(*Gestion des consigne de pompage procédé*)
IF RQ_MARCHE_POMPAGE_PROC OR RQ_MARCHE_REGUL_GAZ[1] OR RQ_MARCHE_REGUL_GAZ[2] THEN
	CONS_MODE := PRM_MODE_PUMPING;
	CONS_PRESSURE := PRM_PR_PUMPING;
	CONS_POSITION := PRM_POS_PUMPING;
	CONS_HI_PRESSURE := PRM_PR_HI_PUMPING;
	CONS_LOW_PRESSURE := PRM_PR_LO_PUMPING;
	CONS_TIM_PRESSURE :=  REAL_TO_TIME ( PRM_TIM_PR_PUMPING * 1000);
END_IF

(*Gestion de la consigne pour la ligne de gaz n°1*)
IF RQ_MARCHE_GAZ[1] THEN
	CONS_FLOW_GAZ_1 := PRM_FLOW_GAZ1;
END_IF

(*Gestion de la consigne pour la ligne de gaz n°2*)
IF RQ_MARCHE_GAZ[2] THEN
	CONS_FLOW_GAZ_2 := PRM_FLOW_GAZ2;
END_IF

(*Demande d'arrêt des sources, que si source pas démarrée pour anticipation*)
RQ_STOP_EVAP_S1 := (FM_ETAPE14.Q AND NOT PRM_UTIL_SOURCE1_ANT) OR (FM_ETAPE10.Q AND NOT PRM_UTIL_SOURCE1);
RQ_STOP_EVAP_S2 := (FM_ETAPE14.Q AND NOT PRM_UTIL_SOURCE2_ANT) OR (FM_ETAPE10.Q AND NOT PRM_UTIL_SOURCE2);
RQ_STOP_EVAP_S3 := (FM_ETAPE14.Q AND NOT PRM_UTIL_SOURCE3_ANT) OR (FM_ETAPE10.Q AND NOT PRM_UTIL_SOURCE3);
RQ_STOP_EVAP_S4 := (FM_ETAPE14.Q AND NOT PRM_UTIL_SOURCE4_ANT) OR (FM_ETAPE10.Q AND NOT PRM_UTIL_SOURCE4);


(*Mise à jour du temps de préparation pour les couches anticipées :
remarque dans le cas de plusieurs sources, elles doivent toutes avoir le même temps de prépa (cf. editeur), mais on prend le max pour sécu*)
IF PRM_UTIL_SOURCE1_ANT THEN
	VAR_TPS_PREPA_ANT1 := PRM_TPS_PREPA_SOURCE1;
	VAR_TPS_PREPA_ANT1_2s := VAR_TPS_PREPA_ANT1 + 5;
ELSE
	VAR_TPS_PREPA_ANT1 := 0;
	VAR_TPS_PREPA_ANT1_2s := 0;
END_IF
IF PRM_UTIL_SOURCE2_ANT THEN
	VAR_TPS_PREPA_ANT2 := PRM_TPS_PREPA_SOURCE2;
	VAR_TPS_PREPA_ANT2_2s := VAR_TPS_PREPA_ANT2 + 5;
ELSE
	VAR_TPS_PREPA_ANT2 := 0;
	VAR_TPS_PREPA_ANT2_2s := 0;
END_IF
IF PRM_UTIL_SOURCE3_ANT THEN
	VAR_TPS_PREPA_ANT3 := PRM_TPS_PREPA_SOURCE3;
	VAR_TPS_PREPA_ANT3_2s := VAR_TPS_PREPA_ANT3 + 5;
ELSE
	VAR_TPS_PREPA_ANT3 := 0;
	VAR_TPS_PREPA_ANT3_2s := 0;
END_IF
IF PRM_UTIL_SOURCE4_ANT THEN
	VAR_TPS_PREPA_ANT4 := PRM_TPS_PREPA_SOURCE4;
	VAR_TPS_PREPA_ANT4_2s := VAR_TPS_PREPA_ANT4 + 5;
ELSE
	VAR_TPS_PREPA_ANT4 := 0;
	VAR_TPS_PREPA_ANT4_2s := 0;
END_IF

(*
(*Les nouvelles épaisseurs se trouvent dans le tableau*)
PRM_EPAISSEUR:= PRM_NEW_EPAISSEUR[STATE_LAYER];
*)

(*calcul du temps restant : version avec vitesse aggrégée théorique (somme des vitesses ds sources utilisées dans l'étape en cours)*)
(*calcul vitesse théorique*)
IF FM_ETAPE12.Q THEN
	VAR_CALCUL_VITESSE_THEORIQUE := PRM_SOURCE1_RATE * BOOL_TO_INT(PRM_UTIL_SOURCE1) +
										PRM_SOURCE2_RATE * BOOL_TO_INT(PRM_UTIL_SOURCE2) +
										PRM_SOURCE3_RATE * BOOL_TO_INT(PRM_UTIL_SOURCE3) +
										PRM_SOURCE4_RATE * BOOL_TO_INT(PRM_UTIL_SOURCE4);
ELSIF OP_RUN.Etape.4 THEN
	VAR_CALCUL_VITESSE_THEORIQUE := 0;
END_IF
IF VAR_CALCUL_VITESSE_THEORIQUE <> 0 THEN
	VAR_TPS_RESTANT_DEPOT := REAL_TO_INT((PRM_EPAISSEUR - I_Global_Thick) / VAR_CALCUL_VITESSE_THEORIQUE);
END_IF


(*temporisation de lissage du bagotage de la vitesse aggrégée si PID pas top, on doit rester inférieur plus de 2s pour lancer la prépa anticipée*)
TIMER_Lancement_Ant_S1.PT := T#1s;
TIMER_Lancement_Ant_S1.IN := (VAR_TPS_RESTANT_DEPOT <= VAR_TPS_PREPA_ANT1_2s) AND TIMER_RAZ_THICKNESS.Q;
TIMER_Lancement_Ant_S1();

TIMER_Lancement_Ant_S2.PT := T#1s;
TIMER_Lancement_Ant_S2.IN := (VAR_TPS_RESTANT_DEPOT <= VAR_TPS_PREPA_ANT2_2s) AND TIMER_RAZ_THICKNESS.Q;
TIMER_Lancement_Ant_S2();

TIMER_Lancement_Ant_S3.PT := T#1s;
TIMER_Lancement_Ant_S3.IN := (VAR_TPS_RESTANT_DEPOT <= VAR_TPS_PREPA_ANT3_2s) AND TIMER_RAZ_THICKNESS.Q;
TIMER_Lancement_Ant_S3();

TIMER_Lancement_Ant_S4.PT := T#1s;
TIMER_Lancement_Ant_S4.IN := (VAR_TPS_RESTANT_DEPOT <= VAR_TPS_PREPA_ANT4_2s) AND TIMER_RAZ_THICKNESS.Q;
TIMER_Lancement_Ant_S4();

(*Lancement de la prépa anticipée seulement si pas de Quartz sous le cache source*)
FM_Prepa_Ant_S1.CLK := 	OP_RUN.Etape.12 AND TIMER_RAZ_THICKNESS.Q AND
						PRM_UTIL_SOURCE1_ANT AND NOT PRM_CTRL_DELAY_SOURCE1 AND
						TIMER_Lancement_Ant_S1.Q;
						(*VAR_TPS_RESTANT_DEPOT <= VAR_TPS_PREPA_ANT1_2s;*)

FM_Prepa_Ant_S2.CLK := 	OP_RUN.Etape.12 AND TIMER_RAZ_THICKNESS.Q AND
						PRM_UTIL_SOURCE2_ANT  AND NOT PRM_CTRL_DELAY_SOURCE2 AND
						TIMER_Lancement_Ant_S2.Q;
						(*VAR_TPS_RESTANT_DEPOT <= VAR_TPS_PREPA_ANT2_2s;*)

FM_Prepa_Ant_S3.CLK := 	OP_RUN.Etape.12 AND TIMER_RAZ_THICKNESS.Q AND
						PRM_UTIL_SOURCE3_ANT AND NOT PRM_CTRL_DELAY_SOURCE3 AND
						TIMER_Lancement_Ant_S3.Q;
						(*VAR_TPS_RESTANT_DEPOT <= VAR_TPS_PREPA_ANT3_2s;*)

FM_Prepa_Ant_S4.CLK := 	OP_RUN.Etape.12 AND TIMER_RAZ_THICKNESS.Q AND
						PRM_UTIL_SOURCE4_ANT AND NOT PRM_CTRL_DELAY_SOURCE4 AND
						TIMER_Lancement_Ant_S4.Q;
						(*VAR_TPS_RESTANT_DEPOT <= VAR_TPS_PREPA_ANT4_2s;*)

FM_Prepa_Ant_S1();
FM_Prepa_Ant_S2();
FM_Prepa_Ant_S3();
FM_Prepa_Ant_S4();


(*Demande de préparation : soit étape 8 sur couche classique (mais pas dans le cas ou elle a été anticipée), soit FM de go anticipation
	(mais que si la source est en étape 0 ou en étape 16, cad arrétée ou cloture finie (sinon le RQ_Evap tombe à l'eau) 
remarque : dans ce cas le var_prepa_lancée est peut etre redondant 

Pas de demande d'anticipation s'il y a un Quartz d'étalonnage de la vitesse de dépôt sous le cache source*)
RQ_PREP_S1 := (FM_ETAPE10.Q AND PRM_UTIL_SOURCE1 AND NOT PRM_ANTICIPATION_COUCHE)
					OR (FM_Prepa_Ant_S1.Q AND NOT  VAR_Prepa_S1_Lancee AND NOT PRM_CTRL_DELAY_SOURCE1
						AND I_SOURCE1_ARRET );

RQ_PREP_S2 := (FM_ETAPE10.Q AND PRM_UTIL_SOURCE2 AND NOT PRM_ANTICIPATION_COUCHE)
					OR (FM_Prepa_Ant_S2.Q AND NOT VAR_Prepa_S2_Lancee AND NOT PRM_CTRL_DELAY_SOURCE2
						AND I_SOURCE2_ARRET);

RQ_PREP_S3 := (FM_ETAPE10.Q AND PRM_UTIL_SOURCE3 AND NOT PRM_ANTICIPATION_COUCHE)
					OR (FM_Prepa_Ant_S3.Q AND NOT VAR_Prepa_S3_Lancee AND NOT PRM_CTRL_DELAY_SOURCE3
						AND I_SOURCE3_ARRET);

RQ_PREP_S4 := (FM_ETAPE10.Q AND PRM_UTIL_SOURCE4 AND NOT PRM_ANTICIPATION_COUCHE)
					OR (FM_Prepa_Ant_S4.Q AND NOT VAR_Prepa_S4_Lancee AND NOT PRM_CTRL_DELAY_SOURCE4
						AND I_SOURCE4_ARRET);



(*variable mise à 1 au premier front montant pour éviter de relancer la prépa si bagotage du temps restant de dépot, remis à 0 en 6 cad apres lecture couche suivante*)
IF FM_Prepa_Ant_S1.Q THEN
	VAR_Prepa_S1_Lancee := TRUE;
ELSIF OP_RUN.Etape.6 OR OP_RUN.Etape.0 THEN
	VAR_Prepa_S1_Lancee := FALSE;
END_IF

IF FM_Prepa_Ant_S2.Q THEN
	VAR_Prepa_S2_Lancee := TRUE;
ELSIF OP_RUN.Etape.6 OR OP_RUN.Etape.0 THEN
	VAR_Prepa_S2_Lancee := FALSE;
END_IF

IF FM_Prepa_Ant_S3.Q THEN
	VAR_Prepa_S3_Lancee := TRUE;
ELSIF OP_RUN.Etape.6 OR OP_RUN.Etape.0 THEN
	VAR_Prepa_S3_Lancee := FALSE;
END_IF

IF FM_Prepa_Ant_S4.Q THEN
	VAR_Prepa_S4_Lancee := TRUE;
ELSIF OP_RUN.Etape.6 OR OP_RUN.Etape.0 THEN
	VAR_Prepa_S4_Lancee := FALSE;
END_IF


(*Lancement évaporation*)
RQ_EVAP_S1 := OP_RUN.Etape.12 AND PRM_UTIL_SOURCE1;
RQ_EVAP_S2 := OP_RUN.Etape.12 AND PRM_UTIL_SOURCE2;
RQ_EVAP_S3 := OP_RUN.Etape.12 AND PRM_UTIL_SOURCE3;
RQ_EVAP_S4 := OP_RUN.Etape.12 AND PRM_UTIL_SOURCE4;

(*Défaut de lecture d'une étape*)
DEF_READ_LAYER.VAL1 := UINT_TO_STRING(STATE_LAYER);
DEF_READ_LAYER.CONDITION := OP_RUN.Etape.20;
DEF_READ_LAYER();

(*Défaut de lecture d'une étape anticipée*)
DEF_READ_LAYER_ANT.VAL1 := UINT_TO_STRING(STATE_LAYER + 1);
DEF_READ_LAYER_ANT.CONDITION := OP_RUN.Etape.21;
DEF_READ_LAYER_ANT();

(*Défaut time out programmation XTC*)
DEF_PROG_QZ.CONDITION := OP_RUN.Etape.9;
DEF_PROG_QZ.DELAY := T#45s;
DEF_PROG_QZ();

(*Défaut time out raz epaisseur controleur XTC*)
DEF_RAZ_QZ.CONDITION := OP_RUN.Etape.11;
DEF_RAZ_QZ.DELAY := T#20s;
DEF_RAZ_QZ();

(*Défaut de passage en STOP du contrôleur de dépôt pendant l'évaporation*)
DEF_CONTROLLER_STOPPED.CONDITION := OP_RUN.Etape.12 AND I_CONTROLEUR_PHASE = 'Deposit' AND  I_Controleur_Stopped;
DEF_CONTROLLER_STOPPED.DELAY:= T#20s;
DEF_CONTROLLER_STOPPED();

(*
(*Défaut de panne quartz générale*)
DEF_QF.CONDITION := I_PC_QUARTZ.STATE_Qz_general_failure AND NOT OP_RUN.Etape.0;
DEF_QF.VAL1 := USINT_TO_STRING(I_PC_QUARTZ.STATE_QF_code);
DEF_QF;
*)

(*reset des ordres*)
IF RCP_NEXT_LAYER AND M_NEXT_LAYER THEN
	M_NEXT_LAYER:=FALSE;
END_IF;


STATE_RATE_AGREGATE := I_Global_Rate;			(*vitesse globale renvoyé par le contrôleur*)
STATE_THICKNESS_AGREGATE  := I_Global_Thick;	(*epaisseur globale renvoyé par le contrôleur*)

STATE_END_OF_LAYER := OP_RUN.Etape.13;
STATE_EVAP := OP_RUN.Etape.12;

IF OP_RUN.Etape.17 THEN
	VAR_Loop_In_Process:= TRUE;
ELSIF OP_RUN.Etape.4 THEN
	VAR_Loop_In_Process:= FALSE;
END_IF

(*Sorties contrôleur*)
OUT_RAZ_THICK_CONTROLEUR:= OP_RUN.Etape.11 AND (NOT I_MODE_REPRISE OR NOT VAR_MEM_LAYER_INTERRUPTED) AND NOT VAR_MEM_COUCHE_TERMINEE;
OUT_RESET_CONTROLEUR:= OP_RUN.Etape.3;
OUT_STOP_CONTROLEUR:= OP_RUN.Etape.2 OR OP_RUN.Etape.13;


IF  OP_RUN.Etape.10 AND (NOT I_MODE_REPRISE OR NOT VAR_MEM_LAYER_INTERRUPTED) THEN
	VAR_MEM_RAZ_THICKNESS := FALSE;
END_IF;
TIMER_RAZ_THICKNESS.PT := T#3s;
TIMER_RAZ_THICKNESS.IN := VAR_MEM_RAZ_THICKNESS;
TIMER_RAZ_THICKNESS();

ACTION RUN_PROCESS:
(*GRAFCET EXECUTION PROCEDE*)
(* initialisation du grafcet*)

OP_RUN(
	N_STEP_OP_OK:=15,
	N_STEP_OP_NOK:= 0);

(* initialisation du grafcet*)
IF 		OP_RUN.Etape = 0 THEN
				OP_RUN.Etape.0 := TRUE;
(*repositionnement sur étape 0*)
ELSIF  NOT I_ON THEN
				OP_Run.Etape:= 0;			(*RAZ grafcet*)
				OP_Run.Etape.0:=TRUE;
(*Repositionnement sur demande fin de couche*)
ELSIF (OP_RUN.Etape.6 OR OP_RUN.Etape.7 OR OP_RUN.Etape.9 OR OP_RUN.Etape.10 OR OP_RUN.Etape.11 OR OP_RUN.Etape.12) AND
		(RCP_NEXT_LAYER)  THEN
				(*si evaporation en cours sur les sources*)
				IF  (OP_RUN.Etape.10 OR OP_RUN.Etape.11 OR OP_RUN.Etape.12) THEN
					RQ_NEXT_LAYER := TRUE; 	(*demande de fin de couche au bloc de gestion des sources*)
				END_IF
				I_MODE_REPRISE := FALSE;
				VAR_MEM_COUCHE_TERMINEE := TRUE;
				(*VAR_Cpt_Boucle:=1;*)	(*RAZ du compteur de boucle*)
				OP_RUN.Etape := 0;
				OP_RUN.Etape.13 := TRUE;
(*étape 0-1 attente ordre execution de l'empilement*)
ELSIF OP_RUN.etape.0 AND I_ON THEN
				OP_RUN.Etape.1 	:=TRUE;
				OP_RUN.Etape.0 	:=FALSE;
(*étape 1-2 *)
ELSIF	OP_RUN.Etape.1 AND NOT I_MODE_REPRISE THEN
				VAR_MEM_LAYER_INTERRUPTED  := FALSE;
				VAR_MEM_COUCHE_TERMINEE := FALSE;
				VAR_MEM_PREP_OPT_TERMINEE := FALSE;
				VAR_Cpt_Boucle:= 1;
				STATE_LAYER:= 1;
				OP_RUN.Etape.2:=TRUE;
				OP_RUN.Etape.1:=FALSE;
(*étape 1-2*)
ELSIF OP_RUN.Etape.1 AND
				(NOT VAR_MEM_LAYER_INTERRUPTED AND I_MODE_REPRISE)
				THEN (*STOP et RESET si mode reprise et pas couche interrompue*)
				OP_RUN.Etape.2:= TRUE;
				OP_RUN.Etape.1:= FALSE;
(*étape 1-4 *)
ELSIF	OP_RUN.Etape.1 AND
				(VAR_MEM_LAYER_INTERRUPTED  AND I_MODE_REPRISE)
				THEN (*Pas de STOP ni de RESET si mode reprise et couche interrompue*)
				OP_RUN.Etape.4:=TRUE;
				OP_RUN.Etape.1:=FALSE;

(*etape 2-3*)
ELSIF OP_RUN.Etape.2  AND TIMER_Stop_Controller.Q(*AND I_ACTION_CONTROLEUR_OK*) THEN
				OP_RUN.Etape.3:=TRUE;
				OP_RUN.Etape.2:=FALSE;

(*etape 3-4*)
ELSIF OP_RUN.Etape.3
				AND TIMER_Reset_Controller.Q (*AND I_ACTION_CONTROLEUR_OK*) AND I_CONTROLEUR_PHASE = 'Ready' THEN		(*IC6 à l'état READY si la RAZ empilement à été effectué *)
				OP_RUN.Etape.4:=TRUE;
				OP_RUN.Etape.3	:=FALSE;

(*etape 4-20*)
ELSIF OP_RUN.Etape.4 AND
				(TIMER_TIMEOUT.Q OR I_LAYER_LOADING_NOK) THEN
				OP_RUN.Etape.20:=TRUE;
				OP_RUN.Etape.4	:=FALSE;

(*etape 4-5*)
ELSIF OP_RUN.Etape.4 AND I_LAYER_LOADING_OK THEN
				OP_RUN.Etape.5		:=TRUE;
				OP_RUN.Etape.4		:=FALSE;

(*etape 5-21*)
ELSIF OP_RUN.Etape.5 AND
				(TIMER_TIMEOUT_ANT.Q OR I_LAYER_ANT_LOADING_NOK) THEN
				OP_RUN.Etape.21 := TRUE;
				OP_RUN.Etape.5 := FALSE;

(*etape 5-6*)
ELSIF OP_RUN.Etape.5 AND (I_LAYER_ANT_LOADING_OK OR I_NO_MORE_LAYER_ANT) THEN	(*Couche anticipée chargé ou pas de couche anticipée*)
				OP_RUN.Etape.6 := TRUE;
				OP_RUN.Etape.5 := FALSE;

(*etape 6-7*)
ELSIF OP_RUN.Etape.6 AND
				((I_ROTATION_PS_OK AND NOT I_NO_ROTATION_PS) OR (I_STOP_ROT_PS_OK AND I_NO_ROTATION_PS))
				AND ((I_STOP_TILT_PS_OK AND I_MODE_TILT = 2) OR (I_MODE_TILT = 1))
				AND I_DOME_IN_POSITION
				AND (
				(I_MARCHE_CHAUFFAGE_OK AND (PRM_MODE_CHAUFFAGE = 1)
						AND (I_STAB_CHAUFFAGE_OK OR NOT PRM_WAIT_STAB_TEMP)
				 )
				OR
				(I_ARRET_CHAUFFAGE_OK AND (PRM_MODE_CHAUFFAGE = 0))
				OR (PRM_MODE_CHAUFFAGE = 2)
				)
				AND(( I_ARRET_GAZ1_OK OR VAR_Util_Gaz[1]) AND (I_ARRET_GAZ2_OK OR VAR_Util_Gaz[2]))
				THEN
				OP_RUN.Etape.7:=TRUE;
				OP_RUN.Etape.6:= FALSE;

(*etape 7-9*)
ELSIF OP_RUN.Etape.7 AND (
				(I_MARCHE_IAD_OK AND PRM_OP_UTIL_IAD) OR
				(I_ARRET_IAD_OK AND NOT PRM_OP_UTIL_IAD) OR NOT CONF_IAD
				)
				AND I_TILT_PS_OK
				AND NOT I_MODE_REPRISE
				THEN
				OP_RUN.Etape.9:=TRUE;
				OP_RUN.Etape.7:=FALSE;

(*etape 7-10 - On ne recharge pas les paramètres dans l'XTC en cas de reprise*)
ELSIF OP_RUN.Etape.7 AND (
				(I_MARCHE_IAD_OK AND PRM_OP_UTIL_IAD) OR
				(I_ARRET_IAD_OK AND NOT PRM_OP_UTIL_IAD) OR NOT CONF_IAD
				)
				AND I_TILT_PS_OK
				AND I_MODE_REPRISE
				THEN
				OP_RUN.Etape.10:=TRUE;
				OP_RUN.Etape.7:=FALSE;

(*Etape 9-10*)
ELSIF OP_RUN.Etape.9 AND I_PROG_CONTROLEUR_OK THEN		(*Programmation contrôleur ok*)
				OP_RUN.Etape.10:=TRUE;
				OP_RUN.Etape.9:=FALSE;

(*Etape 10-11*)
ELSIF OP_RUN.Etape.10
	    AND (I_PREP_SOURCE1_OK OR (NOT PRM_UTIL_SOURCE1 AND I_STOP_EVAP1_OK))
	    AND (I_PREP_SOURCE2_OK OR (NOT PRM_UTIL_SOURCE2 AND I_STOP_EVAP2_OK))
	    AND (I_PREP_SOURCE3_OK OR (NOT PRM_UTIL_SOURCE3 AND I_STOP_EVAP3_OK))
	    AND (I_PREP_SOURCE4_OK OR (NOT PRM_UTIL_SOURCE4 AND I_STOP_EVAP4_OK))
	THEN
				OP_RUN.Etape.11:=TRUE;
				OP_RUN.Etape.10:=FALSE;

(*Demande RAZ épaisseur si pas de mode reprise*)
(*Etape 11-12*)
ELSIF OP_RUN.Etape.11  AND
				(*On vérifie que l'épaisseur à bien été remis à 0*)
				((I_Global_Thick <= 0.1) OR
				(VAR_MEM_LAYER_INTERRUPTED  AND I_MODE_REPRISE) OR
				(VAR_MEM_COUCHE_TERMINEE AND I_MODE_REPRISE)
				)
				AND TIMER_RAZ_EPAISSEUR.Q
				THEN
				(*on déclenche la temporisation aprés RAZ épaisseur*)
				IF (I_Global_Thick<= 0.1) THEN
					VAR_MEM_RAZ_THICKNESS := TRUE;
				END_IF
				VAR_MEM_LAYER_INTERRUPTED := TRUE;
				OP_RUN.Etape.12:=TRUE;
				OP_RUN.Etape.11:=FALSE;

(*Etape 12-13 épaisseur atteinte et tempo de validation de remise à 0 de l'épaisseur*)
ELSIF OP_RUN.Etape.12  AND
			((I_END_DEPOT OR VAR_MEM_COUCHE_TERMINEE) AND TIMER_RAZ_THICKNESS.Q) THEN
				I_MODE_REPRISE := FALSE;
				VAR_MEM_LAYER_INTERRUPTED := FALSE;
				VAR_MEM_COUCHE_TERMINEE := TRUE;
				OP_RUN.Etape.13:=TRUE;
				OP_RUN.Etape.12:=FALSE;

(*Cloture des sources*)
(*Etape 13-16*)
ELSIF OP_RUN.Etape.13
	    AND (I_CLOT_SOURCE1_OK OR NOT PRM_UTIL_SOURCE1
				OR PRM_UTIL_SOURCE1_ANT OR PRM_UTIL_SOURCE2_ANT OR PRM_UTIL_SOURCE3_ANT OR PRM_UTIL_SOURCE4_ANT)
	    AND (I_CLOT_SOURCE2_OK OR NOT PRM_UTIL_SOURCE2
				OR PRM_UTIL_SOURCE1_ANT OR PRM_UTIL_SOURCE2_ANT OR PRM_UTIL_SOURCE3_ANT OR PRM_UTIL_SOURCE4_ANT)
	    AND (I_CLOT_SOURCE3_OK OR NOT PRM_UTIL_SOURCE3
				OR PRM_UTIL_SOURCE1_ANT OR PRM_UTIL_SOURCE2_ANT OR PRM_UTIL_SOURCE3_ANT OR PRM_UTIL_SOURCE4_ANT)
	    AND (I_CLOT_SOURCE4_OK OR NOT PRM_UTIL_SOURCE4
				OR PRM_UTIL_SOURCE1_ANT OR PRM_UTIL_SOURCE2_ANT OR PRM_UTIL_SOURCE3_ANT OR PRM_UTIL_SOURCE4_ANT)
	    AND (((I_ARRET_REGUL_GAZ_OK[1] AND I_MARCHE_POMPAGE_SEC_OK)  OR NOT (PRM_MODE_PUMPING = 2)) OR ((I_ARRET_REGUL_GAZ_OK[2] AND I_MARCHE_POMPAGE_SEC_OK)  OR NOT (PRM_MODE_PUMPING = 3)))
		THEN
				STATE_LAYER := STATE_LAYER +1;
				(*RAZ des flags*)
				VAR_MEM_LAYER_INTERRUPTED := FALSE;
				VAR_MEM_COUCHE_TERMINEE := FALSE;
				OP_RUN.Etape.16:=TRUE;
				OP_RUN.Etape.13:=FALSE;

(*Boucle à effectuer*)
(*Etape 16-17*)
ELSIF OP_RUN.Etape.16
		AND (PRM_LOOP AND ((STATE_LAYER = PRM_LOOP_LAST_LAYER +1) AND (VAR_Cpt_Boucle < PRM_NB_LOOP)))
			THEN
				STATE_LAYER := PRM_LOOP_FIRST_LAYER;
				VAR_Cpt_Boucle:= VAR_Cpt_Boucle + 1;
				OP_RUN.Etape.17:= TRUE;
				OP_RUN.Etape.16:= FALSE;

(*Pas de boucle à effectuer ou nombre de boucle OK*)
(*Etape 16-2*)
ELSIF OP_RUN.Etape.16
		AND ( NOT PRM_LOOP OR NOT (VAR_Cpt_Boucle > PRM_NB_LOOP))  THEN
				OP_RUN.Etape.2	:= TRUE;
				OP_RUN.Etape.16	:= FALSE;
(*
(*Chargement du numéro de couche de départ*)
(*Etape 17-6*)
ELSIF OP_RUN.Etape.17
		AND I_LAYER_LOADING_OK THEN
				OP_RUN.Etape.6:= TRUE;
				OP_RUN.Etape.17:= FALSE;
*)
(*
(*Etape 17-20*)
ELSIF OP_RUN.Etape.17 AND
		(TIMER_TIMEOUT.Q OR I_LAYER_LOADING_NOK) THEN
				OP_RUN.Etape.20:= TRUE;
				OP_RUN.Etape.17:= FALSE;
*)

(*Etape 17-2*)
ELSIF OP_RUN.Etape.17 THEN
				OP_RUN.Etape.2:=TRUE;
				OP_RUN.Etape.17:=FALSE;
(*Etape 4-14*)
ELSIF OP_RUN.Etape.4 AND  I_NO_MORE_LAYER THEN
				OP_RUN.Etape.14:=TRUE;
				OP_RUN.Etape.4:=FALSE;

(*Etape 14-15*)
ELSIF OP_RUN.Etape.14 AND  I_STOP_EVAP1_OK AND I_STOP_EVAP2_OK AND I_STOP_EVAP3_OK
		AND I_DOME_IN_POSITION
		AND I_STOP_ROT_PS_OK
		AND I_STOP_TILT_PS_OK
		AND I_ARRET_REGUL_GAZ_OK[1]
		AND I_ARRET_REGUL_GAZ_OK[2]
		AND I_MARCHE_POMPAGE_SEC_OK
		AND I_STOP_EVAP4_OK  AND I_ARRET_GAZ1_OK AND I_ARRET_GAZ2_OK
		AND (I_ARRET_IAD_OK OR NOT CONF_IAD) THEN
				OP_RUN.Etape.15:=TRUE;
				OP_RUN.Etape.14:=FALSE;
END_IF

OP_RUN.POST();
END_ACTION

END_FUNCTION_BLOCK

// ---- POUs/Fonction/FONCTION MODEMARCHE/BLOCK_STEP_BOUCLE.TcPOU
FUNCTION_BLOCK BLOCK_STEP_BOUCLE

VAR_INPUT
	RESET:							BOOL;
	I_ON:							BOOL;
	I_CURRENT_STEP:					UINT;
	PRM_ITER_BOUCLE:				USINT;
	PRM_ETAPE_BOUCLE:				UINT;
END_VAR

VAR_OUTPUT
	STATE_OK:						BOOL;
	AUTOR_STEP:						BOOL;
	STATE_ITER_BOUCLE:				USINT;
	O_NEXT_STEP:					UINT;
	RQ_BOUCLE:						BOOL;
	RQ_SAUT:						BOOL;
END_VAR

VAR
	MEM_BOUCLE:						BOOL;
	MEM_START_BOUCLE:				UINT;
	MEM_STOP_BOUCLE:				UINT;
	FM_ON:							R_TRIG;
END_VAR

(*Autorisation*)
AUTOR_STEP	:=	( (PRM_ITER_BOUCLE = 0) AND (PRM_ETAPE_BOUCLE > I_CURRENT_STEP) ) (*saut sur étape après*)
					OR
					( (PRM_ITER_BOUCLE > 0) AND (PRM_ETAPE_BOUCLE < I_CURRENT_STEP) ) (*boucle sur étape avant*)
					OR
					( NOT MEM_BOUCLE AND ((MEM_START_BOUCLE <> I_CURRENT_STEP) OR (MEM_STOP_BOUCLE <> PRM_ETAPE_BOUCLE)) ); (*pas 2 boucles imbriquées*)

(*Reset fonction hors procédé*)
IF RESET THEN
	MEM_BOUCLE			:=	FALSE;
	MEM_START_BOUCLE	:=	0;
	MEM_STOP_BOUCLE		:=	0;
	STATE_ITER_BOUCLE	:=	0;
	O_NEXT_STEP			:=	0;
	RQ_BOUCLE				:=	FALSE;
	RQ_SAUT				:=	FALSE;
	STATE_OK				:=	FALSE;
END_IF

IF NOT I_ON THEN
	STATE_OK				:=	FALSE;
	RQ_BOUCLE				:=	FALSE;
	RQ_SAUT				:=	FALSE;
END_IF

(*Front montant*)
FM_ON.CLK	:=	I_ON;
FM_ON();

IF FM_ON.Q THEN
	(*Gestion saut*)
	IF PRM_ITER_BOUCLE = 0 THEN
		MEM_BOUCLE			:=	FALSE;
		MEM_START_BOUCLE	:=	0;
		MEM_STOP_BOUCLE		:=	0;
		STATE_ITER_BOUCLE	:=	0;
		O_NEXT_STEP			:=	PRM_ETAPE_BOUCLE;
		RQ_SAUT				:=	TRUE;
		STATE_OK				:=	TRUE;

	(*Gestion boucle*)
	ELSE
		(*Départ boucle*)
		IF MEM_BOUCLE = 0THEN
			MEM_BOUCLE			:=	TRUE;
			MEM_START_BOUCLE	:=	I_CURRENT_STEP;
			MEM_STOP_BOUCLE		:=	PRM_ETAPE_BOUCLE;
			STATE_ITER_BOUCLE	:=	1;
			O_NEXT_STEP			:=	PRM_ETAPE_BOUCLE;
			RQ_BOUCLE				:=	TRUE;
			STATE_OK				:=	TRUE;
		ELSE
			(*Fin boucle*)
			IF MEM_BOUCLE AND (STATE_ITER_BOUCLE >= PRM_ITER_BOUCLE) THEN
				MEM_BOUCLE			:=	FALSE;
				MEM_START_BOUCLE	:=	0;
				MEM_STOP_BOUCLE		:=	0;
				STATE_ITER_BOUCLE	:=	0;
				O_NEXT_STEP			:=	I_CURRENT_STEP + 1;
				STATE_OK				:=	TRUE;
			(*Suite boucle*)
			ELSE
				MEM_BOUCLE			:=	TRUE;
				MEM_START_BOUCLE	:=	I_CURRENT_STEP;
				MEM_STOP_BOUCLE		:=	PRM_ETAPE_BOUCLE;
				STATE_ITER_BOUCLE	:=	STATE_ITER_BOUCLE + 1;
				O_NEXT_STEP			:=	MEM_STOP_BOUCLE;
				RQ_BOUCLE				:=	TRUE;
				STATE_OK				:=	TRUE;
			END_IF
		END_IF
	END_IF
END_IF

END_FUNCTION_BLOCK

// ---- POUs/Fonction/FONCTIONS PUISSANCE/BLOCK_CPT_USURE.TcPOU
FUNCTION_BLOCK BLOCK_CPT_USURE

VAR_INPUT
	I_Machine_prod:				BOOL;				(*Indicateur de machine en process*)
	I_PRE_EVAP_ON:				BOOL;				(*Indicateur début pré-évaporation*)
	I_EVAP_OFF:					BOOL;				(*Indicateur de fin d'évaporation IDLE*)
	I_EVAP_ON:					BOOL;				(*Indicateur de début d'évaporation*)
	I_LAYER_LOAD_OK:			BOOL;				(*Indicateur chargement couche ok*)
	COUNTER_Evap_Time:		BLOCK_CPT_TEMPS;	(*Compteur temps évaporation*)
END_VAR

VAR
	O_Rapport:					BOOL;		(*demande d'édition du rapport de consommation, c'est l'outil externe qui la fait retomber*)

	FM_Prod:					R_TRIG;		(*Front montant de debut de prod*)
	FM_Layer_Load_Ok:			R_TRIG;		(*Front montant de chargement couche ok*)
	FM_Layer:					R_TRIG;		(*Front montant début évaporation*)

	FD_O_Rapport:				F_TRIG;		(*Front descendant de demande d'édition du rapport*)
	FD_Layer:					F_TRIG;		(*Front descendant de fin de couche*)
	FD_Prod:					F_TRIG;		(*Front descendant de fin de prod*)

	VAR_Log_Needed:			BOOL;		(*Indique si un fichier log doit être crée*)
	VAR_Layer_Done:			BOOL;		(*Indique si la couche a été effectué*)

	pt_Compteur:					POINTER TO UDINT;


END_VAR

VAR_OUTPUT
	(*Données du rapport*)
	STATE_User_Login:			STRING[30];	(*Login user ayant lancé la prod*)
	STATE_User_Name:			STRING[30];	(*Nom user ayant lancé la prod*)
	STATE_User_First:			STRING[30];	(*Prénom user ayant lancé la prod*)

	STATE_Process_Name:		STRING;		(*Nom du procédé lancé*)
	STATE_Date_Deb:			DT;			(*Debut du process*)

	STATE_Config:				STRING;		(*Configuration utilisé*)
	STATE_Crucible:				USINT;		(*Numéro du creuset utilisé*)
	STATE_Material:				STRING;		(*Nom du matériau utilisé*)

	STATE_THICK_Consigne:		REAL;		(*Epaisseur saisie par l'utilisateur au début de la recette*)
	STATE_THICK_Obtenue:		REAL;		(*Epaisseur obtenue en fin de couche ou sur arrêt procédé*)

	STATE_Date_Deb_Evap:		DT;			(*Début d'évaporation*)
	STATE_Date_Fin_Evap:		DT;			(*Fin évaporation*)
	STATE_Temps_Depot:			INT;		(*Temps du dépôt*)

END_VAR

(*Gestion du compteur de temps d'évaporation*)
COUNTER_Evap_Time(I_On := I_EVAP_ON);

pt_Compteur:=ADR(COUNTER_Evap_Time.STATE_CPT);

(*Gestion des fronts*)
FM_Prod(clk := I_Machine_prod);


FD_Prod(clk := I_Machine_prod);

FM_Layer(clk := I_PRE_EVAP_ON );
FD_Layer(clk := I_EVAP_OFF);

FM_Layer_Load_Ok(clk := I_LAYER_LOAD_OK);

FD_O_Rapport(clk := O_Rapport);

(*Remise à 0 des valeurs*)
IF FD_O_Rapport.Q THEN
	STATE_Config				:= '';
	STATE_Crucible				:= 0;
	STATE_Material				:= '';
	STATE_THICK_Consigne		:= 0;
	STATE_THICK_Obtenue			:= 0;
END_IF

(*Enregistrement des données en début de process*)
IF FM_Prod.Q THEN
	STATE_User_Login			:=	PRG_USER.ACTU_USER.LOGIN;
	STATE_User_Name				:=	PRG_USER.ACTU_USER.NOM;
	STATE_User_First			:=	PRG_USER.ACTU_USER.PRENOM;

	STATE_Process_Name		:=	EXECPROC.PRM_PROCESS_NAME;
	STATE_Date_Deb			:=	PRG_SEC._date;

END_IF


(*Enregistrement des données liées à l'empilement*)
IF FM_Layer_Load_Ok.Q THEN
	(*CASE MAIN.STEP_EMPILEMENT.PRM_Type_Dome OF
		0:
			STATE_Config	:=	'250';
		1:
			STATE_Config	:=	'350';
		2:
			STATE_Config	:=	'450';
	END_CASE*)
	STATE_Crucible				:= PRG_EVAP.EVAPS1.PRM_NCR;
	STATE_Material				:= PRG_EVAP.CRUCIBLE1.PRM_MAT[STATE_Crucible];
	STATE_THICK_Consigne		:= MAIN.STEP_EMPILEMENT.PRM_EPAISSEUR;
END_IF


(*Enregistrements des données en début de couche*)
IF FM_Layer.Q THEN
	(*RAZ compteur*)
	pt_Compteur^			:= 0;
	VAR_Layer_Done			:= FALSE;
	VAR_Log_Needed			:= TRUE;
	STATE_Date_Deb_Evap		:= PRG_SEC._date;
END_IF


(*Enregistrements des données en fin de couche*)
IF FD_Layer.Q THEN
	STATE_Date_Fin_Evap		:= PRG_SEC._date;
	STATE_THICK_Obtenue		:= MAIN.STEP_EMPILEMENT.STATE_THICKNESS_AGREGATE;
	STATE_Temps_Depot		:= UDINT_TO_INT(COUNTER_Evap_Time.STATE_Cpt);

	(*Levée du bit de demande de création d'un nouveau fichier*)
	O_Rapport				:=	TRUE;
	VAR_Layer_Done			:=	TRUE;
	VAR_Log_Needed			:=	FALSE;
END_IF


(*Enreistrement des données en fin de production si la couche ne s'est pas terminée*)
IF FD_Prod.Q THEN
	IF NOT VAR_Layer_Done AND VAR_Log_Needed THEN
		STATE_Date_Fin_Evap		:= PRG_SEC._date;
		STATE_THICK_Obtenue		:= MAIN.STEP_EMPILEMENT.STATE_THICKNESS_AGREGATE;
		STATE_Temps_Depot		:= UDINT_TO_INT(COUNTER_Evap_Time.STATE_Cpt);
		(*Levée du bit de demande de création d'un nouveau fichier*)
		O_Rapport				:=	TRUE;
		VAR_Log_Needed			:=	FALSE;
	END_IF
END_IF

END_FUNCTION_BLOCK

// ---- POUs/Fonction/FONCTIONS COMPTEUR/BLOCK_CPT_TEMPS.TcPOU
FUNCTION_BLOCK BLOCK_CPT_TEMPS

(* Fonction de compteur temporel d'utilisation  *)
(*Version 2.0 SP BA8-7326 amélioration par l'utilisation du temps CPU*)

VAR_INPUT
	I_On :						BOOL;					(*donne si la fonction appelante est dans l'état marche (true) ou arret (false) *)
	IN:							BOOL;
END_VAR

VAR_OUTPUT

END_VAR

VAR
	VAR_Date_Off:				T_ULARGE_INTEGER;
	VAR_Date_On:				T_ULARGE_INTEGER;
	FP_On:						R_TRIG;					(*front montant de Etat*)
	FD_On:						F_TRIG;
	TIMER_VALID_ON:				TON;
	_GetCpuCounter:				FW_GetCpuCounter;

END_VAR

VAR_INPUT PERSISTENT
	TagXML:				UINT;
	DISABLE:				BOOL;											(*indique que le compteur est desactivé*)
END_VAR

VAR_TEMP

	_TIM1:						T_ULARGE_INTEGER;
	_TIM2:						LREAL;
	VAR1:						UDINT;
	VAR2:						UDINT;
	VAR3: 						UDINT;
	VAR4:						UDINT;
END_VAR
VAR PERSISTENT
	STATE_Cpt:					 UDINT;				(*contient le temps cumulé d'utilisation de la fonction en seconde*)
END_VAR

IF DISABLE THEN
	RETURN;
END_IF

FP_On(clk:=I_On);
FD_On(clk:= I_On);

TIMER_Valid_On(IN := I_ON ,PT := T#10s);

(*sur front montant de l'odre de marche, on mémorise la date et l'heure courante*)
IF FP_On.Q THEN
	_GetCpuCounter(
				dwCpuCntLo=>VAR1,
				dwCpuCntHi=>VAR2
				);

	VAR_Date_On.dwLowPart := UDINT_TO_DWORD(VAR1);
	VAR_DATE_On.dwHighPart := UDINT_TO_DWORD(VAR2);
END_IF;

(*sur le front descendant ou cycliquement, on met à jour la valeur de temps toutes les minutes*)
IF FD_On.Q OR timer_Valid_on.Q THEN
	TIMER_Valid_On(IN := FALSE);
	_GetCpuCounter(
						dwCpuCntLo=>	VAR3  ,
						dwCpuCntHi=>	VAR4
				 );

	VAR_Date_Off.dwLowPart := UDINT_TO_DWORD(VAR3);
	VAR_DATE_Off.dwHighPart := UDINT_TO_DWORD(VAR4);

	_TIM1 := UInt64Sub64(VAR_DATE_OFF,VAR_DATE_ON);
	_TIM2 := UINT64_TO_LREAL(_TIM1) / 10000000;
	STATE_CPT := STATE_CPT + LREAL_TO_UDINT(((_TIM2)));
	VAR_Date_On := VAR_Date_Off;
END_IF;

END_FUNCTION_BLOCK

// ---- POUs/Fonction/FONCTION MODEMARCHE/BLOCK_MODE_MARCHE_V2_0.TcPOU
FUNCTION_BLOCK BLOCK_MODE_MARCHE_V2_0

(* VERSION 1.0 - 04/2010 - SP*)
(* VERSION 1.1 - 10/2010 - SP - ajout des informations machine*)
(* VERSION 1.2 - 07/2011 - HG - ajout gestion évènements, modification contrôle fonctions, demande arrêt cluster*)
(* VERSION 2.0 - 02/2012 - SP - ajout gestion événements, retrait demande arrêt cluster, prise en compte du mode manuel non sécurisé, ajout
						de la gestion de STATE_COLOR pour animation couleur dans IHM beckhoff en fonction du mode de marche
						7326 - BA8*)
(* VERSION 3.0 - 01/2016 - GV - ajout gestion du chargement des paramètres système au démarrage*)
(* VERSION 4.0 - 05/2022 - GV - ajout du mode standby*)
(* VERSION 5.0 - 11/2023 - HG - Ajout DEF_Presence_TrAC et DEF_Presence_ACSoft avec variables associées
								ajout tempo + STATE_Pause_TrAC avant lancement procédé week-end 
								pour dissociation du procédé et procédé week-end dans trac*)

(* BLOCK GESTION DU MODE DE MARCHE*)

VAR_INPUT
	IN_PT1: 				BOOL;		(* ~ (OPC : 1 : available for OPC-clients) *)		(* Entrée TOR présence tension*)
	IN_MM1:					BOOL;		(* ~ (OPC : 1 : available for OPC-clients) *)		(* Entrée TOR machine en marche*)
	IN_MA1T:				BOOL;		(* ~ (OPC : 1 : available for OPC-clients) *)		(* Entrée TOR pressostat air*)
	IN_MA2T:				BOOL;		(* ~ (OPC : 1 : available for OPC-clients) *)		(* Entrée TOR pressostat N2*)
	EN_Auto:				BOOL:=TRUE;										(*Condition d'autorisation de passage en  mode automatique*)
	EN_Manu:				BOOL:=TRUE;										(*Condition d'autorisation de passage en mode manuel*)
	EN_Prod:				BOOL:=TRUE;										(*Condition d'autorisation de passage en mode production*)
	EN_Standby:				BOOL:=TRUE;										(*Condition d'autorisation de passage en mode standby*)
	EN_Inter_Prod:			BOOL:=TRUE;										(*Condition d'autorisation d'interruption de la production*)
	EN_Reprise_Prod:		BOOL:=TRUE;										(*Condition d'autorisation de reprise de la production*)

	I_Init_OK:				BOOL:=TRUE;										(*information initialisation de la machine ok*)
	I_Param_OK:				BOOL:=TRUE;										(*information de chargement des paramètres système ok*)
	I_Prep_Prod_OK:			BOOL:=TRUE;										(*information préparation production ok*)
	I_PROCEDE_ok:			BOOL:=TRUE;										(*indique que le procédé est terminé normallement*)
	I_ARRET_PROCEDE_OK:		BOOL:=TRUE;										(*indique que l'arrêt procédé est ok*)
	I_INTER_PROD_OK:		BOOL:=TRUE;										(*indique que la séquence d'interruption procédé a été exécutée*)
	I_def_stop:				BOOL;											(*Condition d'arrêt sur défaut*)
	I_Standby_Ok:			BOOL:=TRUE;										(*Information mise en standby ok*)
	I_WakeUp_OK:			BOOL:=TRUE;										(*Information réveille appareils ok*)
	I_PROCEDE_WD_Ok:		BOOL:=TRUE;										(*Procédé week end terminé correctement*)
	I_PROCEDE_WD_Ar:		BOOL:=TRUE;										(*Procédé week end terminé*)
	I_def_inter:			BOOL;											(*Condition d'interruption sur défaut*)
	I_moteur_inter_ok:		BOOL;											(*Moteur de procédé en mode interruption*)

	DEF_Air:					PRCDEF;								(*défaut d'air comprimé*)
	DEF_N2:						PRCDEF;								(*défaut d'azote*)
	EV_Stop_def:				PRCDEF;								(*Evenement arrêt procédé sur défaut*)
	EV_Stop_user:				PRCDEF;								(*Evenement arrêt procédé immédiat sur demande utilisateur*)
	EV_Start_proc:				PRCDEF;								(*Evenement lancement procédé*)
	EV_Stop_Ok:					PRCDEF;								(*Evenement arret normal du procédé*)
	EV_initialisation:			PRCDEF;								(*initialisation de la machine*)
	EV_machine_off:				PRCDEF;								(*arrêt machine*)
	EV_machine_on:				PRCDEF;								(*marche machine*)
	EV_safety_manual_mode:		PRCDEF;								(*passage en mode manuel*)
	EV_auto_mode:				PRCDEF;								(*passage en mode automatique*)
	EV_non_safety_manu_mode:	PRCDEF;								(*désactivation des sécurités en mode manuel*)
	EV_inter_user:				PRCDEF;								(*interruption du procédé*)
	EV_inter_def:				PRCDEF;								(*interruption du procédé sur défaut*)
	EV_reprise:					PRCDEF;								(*Reprise du procédé sur défaut*)
	
	DEF_Presence_TrAC:			PRCDEF;
	DEF_Presence_ACSoft:		PRCDEF;

	COUNTER_Machine_on:			BLOCK_CPT_TEMPS;						(*compteur temps machine en marche*)
	COUNTER_manual_mode:		BLOCK_CPT_TEMPS;						(*compteur temps machine en mode manuel*)
	COUNTER_auto_mode:			BLOCK_CPT_TEMPS;						(*compteur temps machine en mode automatique*)
	COUNTER_production:			BLOCK_CPT_TEMPS;						(*compteur temps machine en production*)

	Etape:						UDINT;			(*étape du grafcet*)
	
	(*Variable procédé weekend*)
	PRM_EXEC_PROC_WEEKEND:		BOOL;	(*Exécution du procédé week end en fin de production*)
	
END_VAR

VAR_INPUT PERSISTENT
	CONF_Name:				STRING;		(* ~ (OPC : 1 : available for OPC-clients) *)		(*nom de la machine*)
	CONF_SerialNumber:		STRING(20);	(* ~ (OPC : 1 : available for OPC-clients) *)		(*N° de série*)
	CONF_Customer:			STRING;		(* ~ (OPC : 1 : available for OPC-clients) *)		(*nom du client*)
	CONF_Version:			STRING(10);	(* ~ (OPC : 1 : available for OPC-clients) *)		(*dernière version du logiciel - personnalisation*)
	CONF_VerDate:			STRING(20);	(* ~ (OPC : 1 : available for OPC-clients) *)		(*date de la dernière version*)
	CONF_Author:			STRING(20);	(* ~ (OPC : 1 : available for OPC-clients) *)		(*auteur*)
	CONF_Model:				STRING(20);	(* ~ (OPC : 1 : available for OPC-clients) *)		(*modele de programme et version *)
	CONF_Affaire:			STRING(10);	(* ~ (OPC : 1 : available for OPC-clients) *)		(*N° d'affaire*)

	CONF_No_MA1T:			BOOL;												(*Option pas de pressostat air*)
	CONF_No_MA2T:			BOOL;												(*Option pas de pressostat N2*)
	
	CONF_TrAC:				BOOL;
	CONF_ACSoft:			BOOL;

	(*Entité*)
	IsAssembly:		BOOL;			(*entité : assembly*)
	IdXML:			STRING;			(*nom entité : identifiant pour recherche dans dico*)
	TagXML:			UINT;			(*nom entité : identifiant pour recherche dans dico*)
	IdParent:		STRING;			(*MNEMO de l'appelant*)
	MNEMO:			STRING;			(*MNEMO de l'entité*)
	
	(*Eco mode*)
	CONF_Tps_Inactivite:		TIME;
	CONF_Standby_Auto:			BOOL;			(*indique si le passage en mode standby est automatique après conf_tps_inactivité*)
	CONF_Wafer_Weekend:			INT;			(*numéro de slot utilisé pour process week end (typiquement, +1 par rapport à slot max de la K7)*)
	
	PRM_PROCESS_WEEKEND: 		STRING;	(* ~ (OPC : 1 : available for OPC-clients) *)				(*Chemin et nom du fichier procédé executé*)
	PRM_PROCESS_NAME_WEEKEND: 	STRING;
	PRM_BATCH_WEEKEND:			STRING;	(* ~ (OPC : 1 : available for OPC-clients) *)				(*Identifiant du lot*)
	PRM_RECORD_WEEKEND:			BOOL;	(*Option d'enregistrement du programme de procédé*)
	PRM_LAUNCHER_WEEKEND:		BOOL;	(*Variable pour indiquer au launcher que l'on souhaite sélectionner le procédé weekend*)
END_VAR

VAR_OUTPUT
	STATE_Auto:			BOOL;		(*indicateur de mode automatique*)
	STATE_Manu:			BOOL;		(*indicateur de mode manuel*)
	STATE_Prod:			BOOL;		(*indicateur de mode production*)
	STATE_Wait_Prod:	BOOL;		(*attente lancement production*)
	STATE_Off:			BOOL;		(*indicateur de machine à l'arrêt*)
	STATE_On:			BOOL;		(*indicateur de machine en marche*)
	STATE_Standby:		BOOL;		(*machine en mode standby*)
	STATE_Inter_Prod:	BOOL;		(*indicateur d'interruption en cours*)
	STATE_interrupted:	BOOL;		(*indicateur de procédé interrompu*)
	STATE_Pause_TrAC:	BOOL;		(*indicateur d'état intermédiaire entre procédé terminé et procédé week-end pas encore lancé*)
	STATUS:				UDINT;		(*code d'état*)
	AUTOR_Auto_Ihm:		BOOL;		(*autorisation de passage en mode automatique depuis l'IHM*)
	AUTOR_Manu_Ihm:		BOOL;		(* autorisation de passage en mode manuel depuis l'IHM*)
	AUTOR_Start_Prod_Ihm:	BOOL;		(* autorisation de marche production depuis l'IHM*)
	AUTOR_Stop_Prod_Ihm:	BOOL;		(* autorisation d'arrêt production depuis l'IHM*)
	AUTOR_Standby_Ihm:		BOOL;		(* autorisation de passage en mode standby depuis l'IHM*)
	AUTOR_Repris_Prod_ihm:	BOOL;		(* autorisation de reprise de la production*)
	AUTOR_Inter_Prod_ihm:	BOOL;		(* autorisation d'interruption de la production*)

	STATE_Color:			DWORD;	(*code couleur en fonction du mode de marche*)

	RQ_Ctrl_Plc:			BOOL;		(*demande de contrôle PLC*)
	RQ_Ctrl_Ihm:			BOOL;		(*demande de contrôle IHM*)
	RQ_Init:				BOOL;		(*demande d'exécution de la séquence d'initialisation*)
	RQ_Write_Param:			BOOL;		(*demande d'écriture des paramètres système*)
	RQ_Prep_Prod:			BOOL;		(*demande d'exécution de la séquence de preparation de la production*)
	RQ_Start_Prod:			BOOL;		(*demande d'exécution de la séquence marche production*)
	RQ_Stop_Prod:			BOOL;		(*demande d'exécution de la séquence d'arrêt production - tous les procédés en cours*)
	RQ_Inter_Prod:			BOOL;		(*Demande d'interruption des procédés*)
	RQ_Standby:				BOOL;		(*demande d'éxécution de la séquence de mise en standby*)
	RQ_Start_Proc_WeekEnd:	BOOL;
END_VAR
VAR
	M_Auto:					BOOL;		(* ordre IHM de passage en mode auto*)
	M_Manu:					BOOL;		(* ordre IHM de passage en mode auto*)
	M_Start_Prod:			BOOL;		(* ordre IHM de lancement de la production*)
	M_Stop_Prod:			BOOL;		(* ordre IHM d'arrêt immédiat de la production*)
	M_inter_Prod:			BOOL;		(* ordre IHM d'interruption de procédé*)
	M_Reprise_Prod:			BOOL;		(* ordre IHM de reprise de procédé*)
	M_Standby:				BOOL;		(* ordre IHM de passage en mode standby*)
	M_End_Standby:			BOOL;		(* ordre IHM de fin de mode standby (passage en auto, si on a le EN_AUTO)*)
	RCP_Auto:				BOOL;
	RCP_Manu:				BOOL;
	RCP_Start_Prod:			BOOL;
	RCP_Stop_Prod:			BOOL;
	RCP_Inter_Prod:			BOOL;
	RCP_Reprise_Prod:		BOOL;
	RCP_Standby:			BOOL;
	RCP_End_Standby:		BOOL;
	FM_etape6:				R_TRIG;
	FM_etape5:				R_TRIG;
	FD_etape6:				F_TRIG;
	Cancel_Process_Weekend: BOOL;
	TIMER_Pause_TrAC:		TON;
END_VAR
VAR_IN_OUT
	PING_TRAC:				BOOL;
	PING_ACSoft:			BOOL;
END_VAR

VAR_EXTERNAL
	MANUAL_SAFETY_OFF: BOOL;
END_VAR

DEF_Air.IdXML					:=	'0';
DEF_Air.TagXML					:=	1;

DEF_N2.IdXML					:=	'0';
DEF_N2.TagXML					:=	2;

EV_Stop_def.IdXML				:=	'0';
EV_Stop_def.TagXML				:=	9;
EV_Stop_def.Groupe				:=	3;

EV_Stop_user.IdXML				:=	'0';
EV_Stop_user.TagXML				:=	10;
EV_Stop_user.Groupe				:=	3;

EV_Start_proc.IdXML				:=	'0';
EV_Start_proc.TagXML			:=	11;
EV_Start_proc.Groupe			:=	3;

EV_Stop_Ok.IdXML				:=	'0';
EV_Stop_Ok.TagXML				:=	12;
EV_Stop_Ok.Groupe				:=	3;

EV_initialisation.idXML			:=	'0';
EV_initialisation.TagXML 		:=	20;
EV_initialisation.Groupe 		:= 	3;

EV_machine_off.IdXML			:=	'0';
EV_machine_off.TagXML 			:=	17;
EV_machine_off.Groupe 			:=	3;

EV_machine_on.IdXML				:=	'0';
EV_machine_on.TagXML			:=	16;
EV_machine_on.Groupe			:=	3;

EV_safety_manual_mode.IdXML		:=	'0';
EV_safety_manual_mode.TagXML	:=	18;
EV_safety_manual_mode.Groupe	:=	3;

EV_non_safety_manu_mode.IdXml 	:=	'0';
EV_non_safety_manu_mode.TagXML 	:=	21;
EV_non_safety_manu_mode.Groupe 	:=	3;

EV_auto_mode.IdXML				:=	'0';
EV_auto_mode.TagXML 			:=	19;
EV_auto_mode.Groupe 			:=	3;

EV_inter_def.IdXML				:=	'0';
EV_inter_def.TagXML 			:=	24;
EV_inter_def.Groupe 			:=	3;

EV_inter_user.IdXML				:=	'0';
EV_inter_user.TagXML 			:=	25;
EV_inter_user.Groupe 			:=	3;

EV_reprise.IdXML				:=	'0';
EV_reprise.TagXML 				:=	26;
EV_reprise.Groupe 				:=	3;

DEF_Presence_TrAC.IdXML			:=	'0';
DEF_Presence_TrAC.TagXML		:=	50;
DEF_Presence_ACSoft.IdXML		:=	'0';
DEF_Presence_ACSoft.TagXML		:=	51;

COUNTER_machine_on.TagXML 		:=	2;
COUNTER_manual_mode.TagXML		:=	3;
COUNTER_auto_mode.TagXML 		:=	4;
COUNTER_production.TagXML		:=	5;

(*reception des ordres*)
RCP_Auto						:=	M_Auto;
RCP_Manu						:=	M_Manu;
RCP_Start_Prod					:=	M_Start_Prod;
RCP_Stop_Prod					:=	M_Stop_Prod;
RCP_Inter_Prod					:=	M_Inter_Prod;
RCP_Reprise_Prod				:=	M_reprise_Prod;
RCP_Standby						:=	M_Standby;
RCP_End_Standby					:=	M_End_Standby;

IF RCP_Stop_Prod THEN
	Cancel_Process_Weekend := TRUE;
END_IF

(*Evenement arrêt procédé sur défaut *)
EV_Stop_DEF.CONDITION	:= ((Etape.8 OR Etape.7 OR etape.12 OR etape.13 OR etape.24) AND I_Def_Stop);
EV_Stop_DEF();
(*arret production sur demande utilisateur*)
EV_Stop_User.CONDITION	:=	(Etape.8 OR Etape.7 OR etape.12 OR etape.13 OR etape.24) AND RCP_Stop_Prod;
EV_Stop_User();
(*arret normal procédé*)
EV_Stop_Ok.CONDITION	:=  ((Etape.8 OR Etape.24) AND I_PROCEDE_ok);
EV_Stop_Ok();
(*evenement mise en mode production*)
EV_Start_proc.CONDITION	:=  (Etape.6 AND EN_Prod AND RCP_Start_Prod);
EV_Start_proc();
(*evenement initialisation*)
EV_initialisation.CONDITION := etape.5;
EV_initialisation();
(*evenement arrêt machine*)
EV_machine_off.CONDITION  := NOT IN_MM1;
EV_machine_off();
(*evenement marche machine*)
EV_machine_on.CONDITION := IN_MM1;
EV_machine_on();
(*evenement passage en mode manuel sécurisé*)
EV_safety_manual_mode.CONDITION := etape.10 AND NOT MANUAL_SAFETY_OFF ;
EV_safety_manual_mode();
(*evenement passage en mode auto*)
EV_auto_mode.CONDITION := etape.6 OR etape.7 OR etape.8 OR etape.11 OR etape.12 OR etape.13 OR etape.14;
EV_auto_mode();
(*evenement désactivation des sécurités en mode manuel*)
EV_non_safety_manu_mode.CONDITION  := etape.10 AND MANUAL_SAFETY_OFF;
EV_non_safety_manu_mode();
(*Evenement d'interruption sur demande utilisateur*)
EV_inter_user.CONDITION := etape.8 AND RCP_Inter_Prod AND EN_Inter_Prod ;
EV_inter_user();
(*Evenement d'interruption sur reprise*)
EV_inter_def.CONDITION := Etape.8 AND I_def_inter;
EV_inter_def();
(*Evenement de reprise aprés interruption*)
EV_reprise.CONDITION := Etape.13 AND RCP_Reprise_Prod AND EN_Reprise_Prod;
EV_reprise();

IF NOT Etape.10 THEN
	MANUAL_SAFETY_OFF := FALSE;
END_IF

(*Gestion des compteurs*)
COUNTER_machine_on(I_On := IN_MM1);
COUNTER_manual_mode(I_On := Etape.10);
COUNTER_auto_mode(I_on:= etape.6);
COUNTER_production(I_on:=etape.7 OR etape.8 OR etape.9);

(*scrutation du graphe*)
GRAPHE();

(*gestion temporisation*)
TIMER_Pause_TrAC.IN	:=	etape.22;
TIMER_Pause_TrAC.PT	:=	T#5S;
TIMER_Pause_TrAC();

(*gestion des états du graphe*)
 IF etape > 0 THEN
	STATUS  :=   LREAL_TO_UINT(LN(UDINT_TO_REAL(etape)) / LN(2));
ELSE
	STATUS := 0;
END_IF

STATE_Auto			:= 	Etape.6 OR Etape.7 OR Etape.8 OR etape.11 OR etape.12 OR etape.13 OR etape.14;
STATE_Manu			:=	Etape.10;
STATE_Prod			:=	Etape.7 OR Etape.8 OR Etape.11 OR Etape.12 OR Etape.13 OR etape.14 OR Etape.22 OR Etape.23 OR Etape.24 OR Etape.25 OR Etape.26;
STATE_Standby		:=	Etape.21;
STATE_Wait_Prod 	:=	Etape.6;
STATE_inter_Prod	:=	Etape.13 OR Etape.12;
STATE_interrupted	:=	Etape.13;
STATE_Pause_TrAC	:=	Etape.22;

(*action en sortie*)
RQ_Init					:=	Etape.5;
RQ_Write_Param			:=	Etape.15;
RQ_Start_Prod			:=	Etape.8;
RQ_Prep_Prod			:=	Etape.7;
RQ_inter_Prod			:= 	Etape.12;
RQ_Stop_Prod			:= 	Etape.11 OR Etape.25;
RQ_Standby				:=	Etape.20;
RQ_Start_Proc_WeekEnd	:=	Etape.24;
STATE_Off				:=	Etape.0 OR Etape.1 OR Etape.2 OR Etape.3;
STATE_On				:=	NOT STATE_Off;

(*demande de controle PLC ou IHM*)
RQ_Ctrl_Ihm	:=	Etape.6 OR Etape.10 OR Etape.13;
RQ_Ctrl_Plc	:=	Etape.5 OR Etape.7 OR Etape.8 OR Etape.11 OR Etape.12 OR Etape.20 OR Etape.21
				OR Etape.22  OR Etape.23 OR Etape.24 OR Etape.25 OR Etape.26 OR NOT IN_MM1;

(*autorisation*)
AUTOR_Auto_Ihm				:=		(Etape.4 OR Etape.10 OR Etape.21) AND EN_Auto;
AUTOR_Manu_Ihm				:=  	(NOT Etape.0 AND NOT Etape.1 AND NOT Etape.2 AND NOT Etape.3 AND NOT Etape.10) AND EN_Manu;
AUTOR_Start_Prod_Ihm		:=		Etape.6 AND EN_Prod AND NOT I_Def_Stop;
AUTOR_Stop_Prod_Ihm			:=		Etape.7 OR Etape.8 OR etape.12 OR etape.13 OR Etape.22 OR Etape.23 OR Etape.24;
AUTOR_Inter_Prod_ihm 		:=		Etape.8 AND EN_Inter_Prod ;
AUTOR_Repris_Prod_Ihm		:=		Etape.13 AND EN_Reprise_Prod  AND NOT I_DEF_INTER;
AUTOR_Standby_Ihm			:=		Etape.6 AND EN_Standby;

(*défaut air*)
DEF_air.CONDITION	:= 	NOT IN_MA1T AND NOT CONF_No_MA1T;
DEF_air.delay		:=	T#5s;
DEF_air();
(*défaut azote*)
DEF_N2.CONDITION	:=	NOT IN_MA2T AND NOT CONF_No_MA2T;
DEF_N2.DELAY		:=	T#5s;
DEF_N2();
(*défaut présence trac*)
DEF_Presence_TrAC.CONDITION	:=	NOT PING_TRAC AND CONF_TrAC;
DEF_Presence_TrAC.DELAY		:=	T#20S;
DEF_Presence_TrAC();
(*défaut présence trac*)
DEF_Presence_ACSoft.CONDITION	:=	NOT PING_ACSoft AND CONF_ACSoft;
DEF_Presence_ACSoft.DELAY		:=	T#60S;
DEF_Presence_ACSoft();


(*reset des ordres de maintenances*)
IF RCP_Auto AND M_Auto THEN
	M_Auto	:=	FALSE;
END_IF;
IF RCP_Manu AND M_Manu THEN
	M_Manu	:=	FALSE;
END_IF;
IF RCP_Start_Prod AND M_Start_Prod THEN
	M_Start_Prod	:=	FALSE;
END_IF;
IF RCP_Stop_Prod AND M_Stop_Prod THEN
	M_Stop_Prod	:=	FALSE;
END_IF;
IF RCP_Inter_Prod  AND M_inter_Prod THEN
	M_Inter_Prod	:=	FALSE;
END_IF;
IF RCP_Reprise_Prod AND M_Reprise_Prod THEN
	M_Reprise_Prod	:=	FALSE;
END_IF;
IF RCP_Standby AND M_Standby THEN
	M_Standby := FALSE;
END_IF
IF RCP_End_Standby AND M_End_Standby THEN
	M_End_Standby := FALSE;
END_IF


(*Gestion des codes couleurs en fonction du mode de marche*)
IF Etape.0 OR etape.1 OR etape.2 OR etape.3 OR etape.4 THEN
	STATE_Color := 16#00FFFFFF; (*blanc*)
ELSIF Etape.5 THEN
	STATE_Color := 16#0FFFFC0; (*bleu*)
ELSIF Etape.7 OR Etape.8 OR Etape.11 THEN
	STATE_Color := 16#0080FF80;	(*vert*)
ELSIF Etape.6 THEN
	STATE_Color := 16#00E0E0E0;	(*gris*)
ELSIF Etape.10 AND NOT MANUAL_SAFETY_OFF THEN
	STATE_Color :=16#080C0FF; (*orange*)
ELSIF Etape.10 AND MANUAL_SAFETY_OFF THEN
	STATE_Color :=16#000000FF; (*rouge*)
END_IF

(*toggle ping*)
PING_TRAC	:=	FALSE;
PING_ACSoft	:=	FALSE;

ACTION GRAPHE:
(*GRAFCET*)
(* initialisation du grafcet*)
IF 		Etape = 0 THEN
				Etape.0 := TRUE;
(*repositionnement sur étape 2*)
ELSIF	NOT  IN_PT1 AND NOT Etape.0 AND NOT Etape.1 AND NOT Etape.2 THEN
				Etape:= 0;			(*RAZ grafcet*)
				Etape.2:=TRUE;
(*repositionnement sur étape 3*)
ELSIF	NOT  IN_MM1 AND NOT Etape.0 AND NOT Etape.1 AND NOT Etape.2 AND NOT Etape.3 THEN
				Etape:= 0;			(*RAZ grafcet*)
				Etape.3:=TRUE;
(*repositionnement sur étape 10 mode manuel*)
ELSIF	RCP_Manu AND EN_Manu  AND NOT Etape.0 AND NOT Etape.1 AND NOT Etape.2 AND NOT Etape.3 AND NOT Etape.10 THEN
				Etape:= 0;			(*RAZ grafcet*)
				Etape.10:=TRUE;
(*étape 0-1*)
ELSIF 	Etape.0 THEN
				Etape.1:=TRUE;
				Etape.0:=FALSE;
(*étape 1-2*)
ELSIF	Etape.1 THEN
				Etape.2:=TRUE;
				Etape.1:=FALSE;
(*étape 2-3*)
ELSIF 	Etape.2
		AND IN_PT1 THEN
				Etape.3:=TRUE;
				Etape.2:=FALSE;
(*étape 3-15*)
ELSIF	Etape.3
		AND IN_MM1 THEN
				Etape.15:=TRUE;
				Etape.3:=FALSE;
(*étape 15-4*)
ELSIF	Etape.15
		AND I_Param_OK THEN
				Etape.4:=TRUE;
				Etape.15:=FALSE;
(*étape 4-5*)
ELSIF 	Etape.4
		AND RCP_Auto
		AND EN_Auto THEN
				Etape.5:=TRUE;
				Etape.4:=FALSE;
(*étape 5-6*)
ELSIF 	Etape.5 AND I_Init_OK THEN
				Etape.6:=TRUE;
				Etape.5:=FALSE;
(*étape 6-7*)
ELSIF 	Etape.6
		AND RCP_Start_Prod
		AND EN_Prod THEN
				Etape.7:=TRUE;
				Etape.6:=FALSE;
(*étape 7-8*)
ELSIF 	Etape.7
		AND I_Prep_Prod_OK THEN
				Etape.8:=TRUE;
				Etape.7:=FALSE;
(*étape 7-11*)
ELSIF 	Etape.7 AND
		(RCP_stop_prod OR
		I_def_stop) THEN
				Etape.11:=TRUE;
				Etape.7:=FALSE;
(*étape 8-11*)
ELSIF	Etape.8 AND
		(RCP_Stop_Prod
		OR I_def_stop
		OR I_PROCEDE_ok) THEN
				Etape.11:=TRUE;
				Etape.8	:=FALSE;
(*étape 8-12*)
ELSIF	Etape.8 AND
		(RCP_Inter_prod
		OR I_def_inter) THEN
				Etape.12:=TRUE;
				Etape.8	:=FALSE;
(*étape 11-6*)
ELSIF	Etape.11 AND
		I_ARRET_PROCEDE_OK AND (NOT PRM_EXEC_PROC_WEEKEND OR Cancel_Process_Weekend) THEN
				Etape.6	:=TRUE;
				Etape.11:=FALSE;
				Cancel_Process_Weekend := FALSE;
(*étape 10-5*)
ELSIF	Etape.10 AND
		RCP_Auto AND
		EN_Auto THEN
				Etape.5	:=TRUE;
				Etape.10:=FALSE;
(*etape 12-13*)
ELSIF 	Etape.12 AND
		I_INTER_PROD_OK AND
		I_MOTEUR_INTER_ok THEN
				Etape.13 := TRUE;
				Etape.12 := FALSE;
(*etape 12-14*)
ELSIF 	Etape.12
		 AND (RCP_Stop_Prod
		OR I_def_stop
		OR I_PROCEDE_ok)  THEN
				Etape.14 := TRUE;
				Etape.12 := FALSE;
(*Etape 14-11*)
ELSIF 	Etape.14 THEN
				etape.11:=TRUE;
				etape.14:=FALSE;
(*etape 13-8 reprise du procédé*)
ELSIF	Etape.13 AND
		RCP_Reprise_Prod AND
		EN_Reprise_Prod THEN
				Etape.8:= TRUE;
				Etape.13:= FALSE;
(*etape 13-11 arrêt du procédé alors que le procédé est interrompu*)
ELSIF	Etape.13 AND (RCP_Stop_Prod
		OR I_def_stop
		OR I_PROCEDE_ok)   THEN
				Etape.11:= TRUE;
				Etape.13:= FALSE;
				
(*étape 6-20 ==> standby*)
ELSIF	Etape.6 AND (RCP_Standby OR MAIN.TIMER_Inactivite.Q) AND EN_Standby THEN
				Etape.20:=TRUE;
				Etape.6:=FALSE;

(*étape 20-21 ==> standby*)
ELSIF	Etape.20 AND I_Standby_Ok THEN
				Etape.21:=TRUE;
				Etape.20:=FALSE;

(*étape 21-27 ==> fin standby*)
ELSIF 	Etape.21  AND (RCP_Auto OR RCP_End_Standby) AND EN_Auto THEN
				Etape.27:=TRUE;
				Etape.21:=FALSE;
				
(*étape 27-5 ==> attente réveille appareil avant init*)
ELSIF	Etape.27 AND I_WakeUp_Ok THEN 
				Etape.5:=TRUE;
				Etape.27:=FALSE;

(*étape 11-22 ==> execution du process week end*)
ELSIF	Etape.11 AND I_ARRET_PROCEDE_OK
				AND PRM_EXEC_PROC_WEEKEND AND NOT Cancel_Process_Weekend THEN
				Etape.22:=TRUE;
				Etape.11:=FALSE;
				Cancel_Process_Weekend:= FALSE;

ELSIF	Etape.22 AND TIMER_Pause_TrAC.Q THEN
				Etape.23:=TRUE;
				Etape.22:=FALSE;

ELSIF	Etape.23 THEN
				Etape.24:=TRUE;
				Etape.23:=FALSE;

(*étape 24-25 procédé week end ok*)
ELSIF	Etape.24 AND I_PROCEDE_WD_Ok THEN
				Etape.25:=TRUE;
				Etape.24:=FALSE;

(*étape 24-26 procédé week end défaut*)
ELSIF	Etape.24 AND (RCP_Stop_Prod OR I_def_stop) THEN
				Etape.26:=TRUE;
				Etape.24:=FALSE;

(*étape 26-25 procédé week end défaut suite*)
ELSIF	Etape.26 AND I_PROCEDE_WD_AR THEN
				Etape.25:=TRUE;
				Etape.26:=FALSE;

(*étape 25-6 fin production week end*)
ELSIF	Etape.25
			AND I_ARRET_PROCEDE_OK
				THEN
				PRM_EXEC_PROC_WEEKEND:=FALSE;
				Etape.6:=TRUE;
				Etape.25:=FALSE;
END_IF;
END_ACTION

END_FUNCTION_BLOCK

// ---- POUs/Fonction/FONCTION MODEMARCHE/BLOCK_INIT_MACHINE.TcPOU
FUNCTION_BLOCK BLOCK_INIT_MACHINE

(*block de gestion d'initialisation d'une machine de type EVA601 sans SAS*)

(****************historique des versions*****************************)
(* Version 1-0 - GV - VERSION INITIALE - 12191 *)
(* Version 1-1 - GV - Demande arrêt XTC si pas en Stop - 13375 - 09/2022*)
(*************************************************************************)


VAR_INPUT
	(*demandes par bloc Mode de Marche*)
	CO_Inter:					BOOL;
	CO_Stop_Prod:				BOOL;
	CO_Init_Prod:				BOOL;
	CO_init:					BOOL;
	OP_init:					BLOCK_G7;

	M_Stop_Procedure:			BOOL;		(*Ordre IHM d'interruption de la procédure d'arrêt*)
	RCP_Stop_Procedure:			BOOL;
                                
	I_STOP_EVAP_OK:				BOOL;
	I_STOP_CONTROLLER_OK:		BOOL;
	I_STOP_EFFLUVAGE_OK:		BOOL;
	I_STOP_GAZ_OK:				BOOL;
	I_STOP_CHAUFFAGE_OK:		BOOL;
	I_STOP_MVTS_OK:				BOOL;
	I_INIT_PRISE_OK:			BOOL;
	I_INIT_POSE_OK:				BOOL;
	I_STOP_IAD_OK:				BOOL;
	I_POMPAGE_SEC_OK:			BOOL;
	I_TH_ATM:					BOOL;
	I_DOOR:						BOOL;
	I_PURGE_EC:				BOOL;
END_VAR
VAR
	FM_Etape1:					R_TRIG;
	FM_Etape2:					R_TRIG;
	FM_Etape3:					R_TRIG;
	FM_Etape4:					R_TRIG;
	FM_Etape5:					R_TRIG;
	FM_Etape6:					R_TRIG;
	FM_Etape7:					R_TRIG;
	FM_Etape8:					R_TRIG;

	I_PURGE_RAH_OK: BOOL;
END_VAR

VAR_OUTPUT
	STATE_OK:					BOOL;
	RQ_STOP_EFFLUVAGE:			BOOL;
	RQ_STOP_CHAUFFAGE:			BOOL;
	RQ_STOP_GAZ:				BOOL;
	RQ_STOP_EVAP:				BOOL;
	RQ_STOP_CONTROLLER:			BOOL;
	RQ_START_PUMP:				BOOL;
	RQ_START_PUMPING:			BOOL;
	RQ_STOP_MVTS:				BOOL;
	RQ_STOP_IAD:				BOOL;
	RQ_INIT_PRISE:				BOOL;
	RQ_INIT_POSE:				BOOL;
                                
	STATE_ABORT:				BOOL;	(*Indique que la procédure d'arrêt est en cours*)

END_VAR
VAR_INPUT PERSISTENT
	IsFunction:		BOOL;			(*entité : fonction*)
	IdXML:			STRING;			(*nom entité : identifiant pour recherche dans dico*)
	TagXML:			UINT;			(*nom entité : identifiant pour recherche dans dico*)
	IdParent:		STRING;			(*MNEMO de l'appelant*)
	MNEMO:			STRING;			(*MNEMO de l'entité*)
END_VAR


VAR
	I:				INT;		(*Variable d'itération*)
END_VAR

(*Scrutation G7*)
ACT_INIT();

FM_etape1(CLK:=OP_init.Etape.1);
FM_etape2(CLK:=OP_init.Etape.2);
FM_etape3(CLK:=OP_init.Etape.3);
FM_etape4(CLK:=OP_init.Etape.4);
FM_etape5(CLK:=OP_init.Etape.5);
FM_etape6(CLK:=OP_init.Etape.6);
FM_etape7(CLK:=OP_init.Etape.7);
FM_etape8(CLK:=OP_init.Etape.8);

RQ_STOP_CONTROLLER := OP_Init.Etape.1 AND NOT I_STOP_CONTROLLER_OK;
RQ_STOP_EVAP := FM_ETAPE1.Q;
RQ_STOP_IAD:= FM_ETAPE2.Q OR FM_ETAPE7.Q;
RQ_STOP_EFFLUVAGE := FM_ETAPE1.Q;
RQ_STOP_CHAUFFAGE := FM_ETAPE1.Q;
RQ_STOP_GAZ := (FM_ETAPE1.Q AND NOT I_PURGE_EC);
RQ_STOP_MVTS := FM_ETAPE1.Q;
RQ_START_PUMP := FM_ETAPE5.Q;
RQ_START_PUMPING := FM_ETAPE6.Q;
RQ_INIT_POSE := FM_ETAPE3.Q AND I_DOOR AND CO_Stop_Prod;
RQ_INIT_PRISE := FM_ETAPE4.Q AND I_DOOR AND CO_Init_Prod;


STATE_OK:=	OP_INIT.OK;

ACTION ACT_INIT:
OP_INIT(
	N_STEP_OP_OK:= 8,
	N_STEP_OP_NOK:= 0);

(*GRAFCET*)
(* initialisation du grafcet*)
IF 		OP_INIT.ETAPE = 0
		THEN
				OP_INIT.ETAPE.0 := TRUE;
(*repositionnement sur étape 0*)
ELSIF	NOT CO_Inter  AND NOT CO_Init AND NOT CO_Stop_Prod AND NOT CO_Init_Prod THEN

				OP_INIT.ETAPE := 0;			(*RAZ grafcet*)
				OP_INIT.ETAPE.0:=TRUE;
(*étape 0-1*)
ELSIF 	OP_INIT.ETAPE.0
		AND (CO_Init
		OR CO_Stop_Prod
		OR CO_Init_Prod
		OR CO_Inter)
		THEN
				OP_INIT.ETAPE.1:=TRUE;
				OP_INIT.ETAPE.0:=FALSE;
(*étape 1-2*)
ELSIF	OP_INIT.Etape.1
		AND I_STOP_EVAP_OK
		AND I_STOP_CONTROLLER_OK
		AND I_STOP_EFFLUVAGE_OK
		AND I_STOP_CHAUFFAGE_OK
		AND (I_STOP_GAZ_OK OR I_PURGE_EC)
	 	AND I_STOP_MVTS_OK
		THEN
				OP_INIT.ETAPE.2:=TRUE;
				OP_INIT.ETAPE.1:=FALSE;
(*étape 2-3*)
ELSIF OP_INIT.Etape.2
		AND I_STOP_IAD_OK THEN
				OP_INIT.Etape.3 := TRUE;
				OP_INIT.Etape.2 := FALSE;
(*étape 3-4*)
ELSIF 	OP_INIT.Etape.3
		AND (I_INIT_POSE_OK OR NOT I_DOOR OR NOT CO_Stop_Prod) THEN
				OP_INIT.Etape.4 := TRUE;
				OP_INIT.Etape.3 := FALSE;
(*étape 4-5*)
ELSIF	OP_INIT.Etape.4
		AND (I_INIT_PRISE_OK OR NOT I_DOOR OR NOT CO_Init_Prod) THEN
				OP_INIT.Etape.5 := TRUE;
				OP_INIT.Etape.4 := FALSE;
(*étape 5-8*)
ELSIF	OP_INIT.Etape.5
		AND I_TH_Atm THEN
				OP_INIT.Etape.8 := TRUE;
				OP_INIT.Etape.5 := FALSE;
(*étape 5-6*)
ELSIF	OP_INIT.Etape.5
		AND NOT I_TH_Atm AND I_DOOR
		THEN
				OP_INIT.Etape.6 := TRUE;
				OP_INIT.Etape.5 := FALSE;
(*étape 6-7*)
ELSIF	OP_INIT.Etape.6
		AND I_POMPAGE_SEC_OK
		THEN
				OP_INIT.Etape.7 := TRUE;
				OP_INIT.Etape.6 := FALSE;
(*étape 7-8*) (*Redemande d'arrêt IAD pour purge d'arrêt si besoin*)
ELSIF	OP_INIT.Etape.7
		AND I_STOP_IAD_OK
		THEN
				OP_INIT.Etape.8 := TRUE;
				OP_INIT.Etape.7 := FALSE;
END_IF
OP_INIT.POST();
END_ACTION

END_FUNCTION_BLOCK

// ---- POUs/Fonction/FONCTION MODEMARCHE/BLOCK_EXEC_PROC.TcPOU
FUNCTION_BLOCK BLOCK_EXEC_PROC

(*block de gestion d'éxécution des procédés d'une machine de type EVA*)

(****************historique des versions*****************************)
(* Version 1-0 - GV - VERSION INITIALE - 9070*)
(* Version 2-0 - GV - 9310 - 01/2016 - Modification gestion PULL_TRAC type lent *)
(* Version 3-0 - HG - 11355 - 03/2019 - Ajout gestion paramètres boucle/saut pour numéro étape à demander à ACSoft 
								+ texte évènement*)
(* Version 4-0 - GV - 13375 - 10/2022 - Modificiation variable PULL_TRAC pour gestion avec nouveau TR'AC*)
(* Version 5-0 - HG - 14035 - 11/2023 - Suppression PULL_TRAC, géré dans BLOCK_MODE_MARCHE V5*)
(*************************************************************************)

VAR_INPUT
	I_ON:						BOOL;					(*Condition de déclenchement du grafcet de marche du procédé*)
	I_PROCESS_LOADING_OK:		BOOL;					(*l'IHM indique que le procédé a été chargé sans erreur*)
	I_PROCESS_LOADING_NOK:		BOOL;					(*L'IHM indique une erreur de chargement du procédé*)
	I_STEP_LOADING_OK:			BOOL;					(*L'IHM indique le chargement de l'étape ok*)
	I_STEP_LOADING_NOK:			BOOL;					(*L'IHM indique le chargement de l'étape nok*)
	I_NO_MORE_STEP:				BOOL;					(*L'IHM indique qu'il n'y a plus d'étape à exécuter*)
	I_INTER_PROC:				BOOL;					(*information d'interruption du procédé en cours*)

	M_LOAD_PROCESS:				BOOL;					(*Demande opérateur de chargement du process*)

	EN_EXEC_STEP:					ARRAY[0..30] OF BOOL;	(*Condition d'autorisation d'exécution des étapes*)
	EN_NEXT_STEP:					ARRAY[0..30] OF BOOL;	(*Condition d'autorisation d'exécution de l'étape suivante*)

	M_NEXT_STEP:					BOOL;

	I_EXEC_STEP_OK:					ARRAY[0..30] OF BOOL;	(*Execution étape ok*)

	(*défaut*)
	DEF_PROCESS_LOADING:		PRCDEF;				(*défaut de chargement du procédé*)
	DEF_STEP_REJECTED:			PRCDEF;				(*défaut d'étape non autorisée*)
	DEF_READ_STEP:				PRCDEF;				(*défaut de lecture d'une étape*)

	(*évenement*)
	EV_LOAD_PROCESS:				PRCDEF;				(*Evenement chargement d'un procédé*)
	EV_LOAD_STEP:					PRCDEF;				(*Evenement chargement d'une étape*)
	EV_STEP_BOUCLE:					PRCDEF;				(*Evenement boucle Xeme itération*)
	EV_NEXT_STEP:					PRCDEF;				(*Evenement de passage à l'étape suivante*)

	PRM_PROCESS: 				STRING;					(* ~ (OPC : 1 : available for OPC-clients) *)				(*Chemin et nom du fichier procédé executé*)
	PRM_PROCESS_NAME: 			STRING;
	PRM_TYPE_ETAPE:				UINT;					(*Type d'étape à exécuter*)
	PRM_BATCH:					STRING;					(* ~ (OPC : 1 : available for OPC-clients) *)				(*Identifiant du lot*)
	PRM_RECORD:					BOOL;					(*Option d'enregistrement du programme de procédé*)
	PRM_NEXT_STEP_EXT:			ARRAY[0..30] OF BOOL;	(*Indique que la fonction fin d'étape anticipée est prise en charge de manière externe*)
	PRM_BOUCLE:					BOOL:=FALSE;			(*Indique que l'étape courante est une boucle : gestion numéro étape suivante*)
	PRM_SAUT:					BOOL:=FALSE;			(*Indique que l'étape courante est un saut : gestion numéro étape suivante*)
	PRM_NEXT_STEP:				UINT;					(*N° d'étape suivante si boucle/saut*)
	I_ITER_BOUCLE:				USINT;					(*Itération courante boucle*)

	OP_RUN:						BLOCK_G7;				(*Grafcet de gestion de l'execution procede*)
END_VAR

VAR_INPUT PERSISTENT
	IsFunction:		BOOL;			(*entité : fonction*)
	IdXML:			STRING;			(*nom entité : identifiant pour recherche dans dico*)
	TagXML:			UINT;			(*nom entité : identifiant pour recherche dans dico*)
	IdParent:		STRING;			(*MNEMO de l'appelant*)
	MNEMO:			STRING;			(*MNEMO de l'entité*)
END_VAR
VAR_OUTPUT
	RQ_EXEC_STEP:					ARRAY[0..30] OF BOOL;
	RQ_LOAD_PROCESS:				BOOL;						(*Demande de chargement du procédé dans l'HM*)
	RQ_READ_STEP:					BOOL;						(*Demande de lecture de l'étape suivante*)
	RQ_FM_EXEC_STEP:				ARRAY[0..30] OF BOOL;		(*Front montant demande de lecture procédé dans l'IHM*)
	STATE_INTERRUPTED:				BOOL;						(*Indicateur de procédé interrompu*)
	STATE_STEP:						UINT;						(*N° d'étape en cours d'exécution*)
	STATE_OK:						BOOL;
	STATUS:							UINT;						(*Etat du grafcet*)
	STATE_STEP_TEXT:				STRING(255);				(*Descriptif de l'étape en cours d'exécution*)
	AUTOR_NEXT_STEP:				BOOL;					(*Autorisation de passage à l'étape suivante*)
	STATE_reprise:					BOOL;						(*indicateurateur de mode reprise en cours*)
	RQ_NEXT_STEP:					BOOL;						(* transmission de l'ordre d'étape suivante au étape complexe*)
	STATE_RECORD:					BOOL;	(* ~ (OPC : 1 : available for OPC-clients) *)

	(*requetes vérification*)
	RQ_Verif_Prog:			BOOL;						(*Demande vérification du programme de procédé*)
END_VAR

VAR
	TIMER_TIMEOUT:				TON;		(*Timer timemout lecture étape*)
	TIMER_RCP_PROCESS:			TP;
	RCP_NEXT_STEP:				BOOL;
	RCP_LOAD_PROCESS:			BOOL;
	FM_ETAPE5:					R_TRIG;
	FM_ETAPE0:					R_TRIG;
	TIMER_RESET_BATCH:			TP;
	FD_TIMER_RESET:				F_TRIG;
	TIMER_RELOAD_PROCESS: 		TP;
END_VAR

DEF_PROCESS_LOADING.IdXML := '0';
DEF_PROCESS_LOADING.TagXML := 27;
DEF_READ_STEP.IdXML := '0';
DEF_READ_STEP.TagXML := 28;
DEF_STEP_REJECTED.IdXML := '0';
DEF_STEP_REJECTED.TagXML := 29;

EV_LOAD_PROCESS.IdXML := '0';
EV_LOAD_PROCESS.TagXML :=30;
EV_LOAD_PROCESS.Groupe := 3;

EV_LOAD_STEP.IdXML := '0';
EV_LOAD_STEP.TagXML :=31;
EV_LOAD_STEP.Groupe := 3;

EV_STEP_BOUCLE.IdXML := '0';
EV_STEP_BOUCLE.TagXML :=41;
EV_STEP_BOUCLE.Groupe := 3;

EV_NEXT_STEP.IdXML :='0';
EV_NEXT_STEP.TagXML :=32;
EV_NEXT_STEP.Groupe := 3;


IdXML :='19';
TagXML := 1;

(*Demande de vérification procédé*)
RQ_Verif_Prog	:=	OP_RUN.Etape.1;

(*Reception des ordres*)
RQ_NEXT_STEP:= FALSE;
RCP_NEXT_STEP:= M_NEXT_STEP;
RQ_NEXT_STEP:=RCP_NEXT_STEP;

RCP_LOAD_PROCESS:= M_LOAD_PROCESS;
TIMER_RCP_PROCESS(IN:=M_LOAD_PROCESS  ,PT:=T#1s);

TIMER_RELOAD_PROCESS(IN:=RCP_LOAD_PROCESS , PT:=T#2s);


(*Evenement de lecture d'une étape*)
EV_LOAD_STEP.VAL1 := UINT_TO_STRING(STATE_STEP);
EV_LOAD_STEP.VAL2 := STATE_STEP_TEXT;
EV_LOAD_STEP.CONDITION := OP_RUN.Etape.2 AND I_STEP_LOADING_OK AND NOT PRM_BOUCLE;
EV_LOAD_STEP();

(*Evenement de lecture d'une étape boucle*)
EV_STEP_BOUCLE.VAL1 := UINT_TO_STRING(STATE_STEP);
EV_STEP_BOUCLE.VAL2 := STATE_STEP_TEXT;
EV_STEP_BOUCLE.VAL3 := USINT_TO_STRING(I_ITER_BOUCLE+1);
EV_STEP_BOUCLE.CONDITION := OP_RUN.Etape.5 AND (I_EXEC_STEP_OK[PRM_TYPE_ETAPE]) AND PRM_BOUCLE;
EV_STEP_BOUCLE();

EV_NEXT_STEP.CONDITION :=OP_RUN.Etape.5
						AND RCP_NEXT_STEP AND AUTOR_NEXT_STEP;
EV_NEXT_STEP();

RUN_PROCESS();


(*Temporisation de time out*)
TIMER_TIMEOUT	(
				PT:=T#5s,
				IN:=OP_RUN.Etape.2
				);

(*Demande de chargement procédé*)
RQ_LOAD_PROCESS		:= 	OP_RUN.Etape.1
						OR (TIMER_RCP_PROCESS.Q AND NOT I_PROCESS_LOADING_OK AND NOT I_PROCESS_LOADING_NOK)  ;
RQ_READ_STEP 			:= 	OP_run.Etape.2;

FM_ETAPE5(CLK:=OP_RUN.Etape.5);
RQ_FM_EXEC_STEP[PRM_TYPE_ETAPE] 		:=	FM_ETAPE5.Q;
RQ_EXEC_STEP[PRM_TYPE_ETAPE]			:=	OP_RUN.Etape.5;
IF NOT RQ_LOAD_PROCESS THEN
	I_PROCESS_LOADING_OK:=FALSE;
	I_PROCESS_LOADING_NOK:=FALSE;
END_IF
IF NOT RQ_READ_STEP THEN
	I_STEP_LOADING_NOK := FALSE;
	I_STEP_LOADING_OK:=FALSE;
	I_NO_MORE_STEP :=FALSE;
END_IF

(*N°d'étape en cours*)
IF OP_RUN.Etape.1 THEN
	STATE_STEP	:=	1;
ELSIF OP_RUN.Etape.6 AND NOT PRM_BOUCLE AND NOT PRM_SAUT THEN
	STATE_STEP := STATE_STEP + 1;
ELSIF OP_RUN.Etape.6 AND (PRM_BOUCLE OR PRM_SAUT) THEN
	STATE_STEP := PRM_NEXT_STEP;
END_IF
STATE_OK:=OP_RUN.OK;
(*Gestion du mode reprise*)
IF OP_RUN.Etape.9 THEN
	STATE_reprise := TRUE;
ELSIF OP_RUN.Etape.0 OR OP_RUN.Etape.6 THEN
	STATE_Reprise:=FALSE;
END_IF

(*interruption procédé*)
STATE_INTERRUPTED	 := 	OP_RUN.Etape.8;
STATUS				 := 	OP_RUN.STATUS;
AUTOR_NEXT_STEP		 :=		EN_NEXT_STEP[PRM_TYPE_ETAPE] AND OP_RUN.Etape.5;


(*Défaut de chargement du procédé*)
DEF_PROCESS_LOADING.CONDITION:=OP_RUN.Etape.12;
DEF_PROCESS_LOADING();
(*Défaut d'étape non autorisés*)
DEF_STEP_REJECTED.VAL1 := UINT_TO_STRING(STATE_STEP);
DEF_STEP_REJECTED.VAL2:=STATE_STEP_TEXT ;
DEF_STEP_REJECTED.CONDITION:=OP_RUN.Etape.7;
DEF_STEP_REJECTED();
(*Défaut de lecture d'une étape*)
DEF_READ_STEP.VAL1 := UINT_TO_STRING(STATE_STEP);
DEF_READ_STEP.CONDITION := OP_RUN.Etape.11;
DEF_READ_STEP();

(*Evenement de chargement d'un procédé*)
EV_LOAD_PROCESS.VAL1 := PRM_PROCESS;
EV_LOAD_PROCESS.VAL2 := PRM_BATCH;
EV_LOAD_PROCESS.CONDITION := OP_RUN.Etape.1 OR ( TIMER_RCP_PROCESS.Q AND I_PROCESS_LOADING_OK)  ;
EV_LOAD_PROCESS();

(*reset des ordres*)
IF RCP_NEXT_STEP AND M_NEXT_STEP THEN
	M_NEXT_STEP:=FALSE;
END_IF;
IF RCP_LOAD_PROCESS AND M_LOAD_PROCESS THEN
	M_LOAD_PROCESS:=FALSE;
END_IF;

STATE_RECORD := PRM_RECORD AND NOT OP_RUN.Etape.0;
FM_ETAPE0(CLK:=OP_RUN.Etape.0);
TIMER_RESET_BATCH( IN:= FM_ETAPE0.Q ,
						PT:= T#5s);

FD_TIMER_RESET(CLK:= TIMER_RESET_BATCH.Q);
IF FD_TIMER_RESET.q  THEN
	PRM_BATCH := '';
END_IF

ACTION RUN_PROCESS:
(*GRAFCET EXECUTION PROCEDE*)
(* initialisation du grafcet*)

OP_RUN(
	N_STEP_OP_OK:=10 ,
	N_STEP_OP_NOK:= 0);

(* initialisation du grafcet*)
IF 		OP_RUN.Etape = 0 THEN
				OP_RUN.Etape.0 := TRUE;
(*interruption du procédé - repositionnement sur étape 8*)
ELSIF NOT OP_RUN.Etape.0 AND I_INTER_PROC THEN
				OP_RUN.Etape := 0;
				OP_RUN.Etape.8:=TRUE;
(*repositionnement sur étape 0*)
ELSIF  NOT I_ON AND NOT OP_RUN.Etape.0 THEN

				OP_Run.Etape:= 0;			(*RAZ grafcet*)
				OP_Run.Etape.0:=TRUE;
(*étape 0-1 attente ordre execution du procede*)
ELSIF OP_RUN.etape.0 AND I_ON  THEN
				OP_RUN.Etape.1 	:=TRUE;
				OP_RUN.Etape.0 	:=FALSE;
(*étape 1-2 chargement procede ok*)
ELSIF	OP_RUN.Etape.1 AND I_PROCESS_LOADING_OK  THEN
				OP_RUN.Etape.2:=TRUE;
				OP_RUN.Etape.1:=FALSE;
(*étape 1-12 chargement procede nok*)
ELSIF	OP_RUN.Etape.1 AND I_PROCESS_LOADING_NOK  THEN
				OP_RUN.Etape.12:=TRUE;
				OP_RUN.Etape.1:=FALSE;
(*etape 2-3*)
ELSIF OP_RUN.Etape.2 AND I_STEP_LOADING_OK THEN
				OP_RUN.Etape.3:=TRUE;
				OP_RUN.Etape.2:=FALSE;
(*etape 2-11*)
ELSIF OP_RUN.Etape.2 AND (TIMER_TIMEOUT.Q OR I_STEP_LOADING_NOK)  THEN
				OP_RUN.Etape.11:=TRUE;
				OP_RUN.Etape.2	:=FALSE;
(*etape 2-10*)
ELSIF OP_RUN.Etape.2 AND I_NO_MORE_STEP THEN
				OP_RUN.Etape.10:=TRUE;
				OP_RUN.Etape.2:= FALSE;
(*etape 3-4*)
ELSIF OP_RUN.Etape.3 THEN
				OP_RUN.Etape.4:=TRUE;
				OP_RUN.Etape.3:= FALSE;
(*etape 4-5*)
ELSIF OP_RUN.Etape.4 AND EN_EXEC_STEP[PRM_TYPE_ETAPE] THEN
				OP_RUN.Etape.5:=TRUE;
				OP_RUN.Etape.4:=FALSE;
(*Etape 4-7*)
ELSIF OP_RUN.Etape.4 AND NOT EN_EXEC_STEP[PRM_TYPE_ETAPE] THEN
				OP_RUN.Etape.7:=TRUE;
				OP_RUN.Etape.4:=FALSE;
(*Etape 5-6*)
ELSIF OP_RUN.Etape.5 AND (I_EXEC_STEP_OK[PRM_TYPE_ETAPE]
						OR (RCP_NEXT_STEP AND AUTOR_NEXT_STEP  AND NOT PRM_NEXT_STEP_EXT[PRM_TYPE_ETAPE])) THEN
				OP_RUN.Etape.6:=TRUE;
				OP_RUN.Etape.5:=FALSE;
(*Etape 6-2*)
ELSIF OP_RUN.Etape.6  THEN
				OP_RUN.Etape.2:=TRUE;
				OP_RUN.Etape.6:=FALSE;
(*Etape 8-9*)
ELSIF OP_RUN.Etape.8  AND NOT I_INTER_PROC THEN
				OP_RUN.Etape.9:=TRUE;
				OP_RUN.Etape.8:=FALSE;
(*Etape 9-2*)
ELSIF OP_RUN.Etape.9   THEN
				OP_RUN.Etape.2:=TRUE;
				OP_RUN.Etape.9:=FALSE;
END_IF

OP_RUN.POST();
END_ACTION

END_FUNCTION_BLOCK

// ---- POUs/Fonction/FONCTION MODEMARCHE/BLOCK_1RUN_1QUARTZ.TcPOU
FUNCTION_BLOCK BLOCK_1RUN_1QUARTZ

VAR_INPUT
	I_Prod:					BOOL;		(*Production en cours*)
	I_Evap:					BOOL;		(*Evaporation en cours - pour mémorisation quartz utilisé*)
	I_CD6T:					BOOL;		(*Demande switch quartz par XTC - pour détection switch pendant evap*)	
	I_QF:					ARRAY[1..12] OF BOOL; (*Mémoire quartz en défaut*)
	M_Mode:					BOOL;		(*activation/désactivation mode 1run = 1quartz*)
	M_RAZ_Quartz:			BOOL;		(*forcage changement des quartz au prochain run - pour sortie mode manuel si nécessaire*)
	I_Current_Quartz:		INT;		(*quartz courant*)
	DEF_Stop_Quartz:		PRCDEF;		(*défaut switch quartz trop nombreux*)
	DEF_No_Quartz:			PRCDEF;		(*défaut pas de quartz pour la production*)
END_VAR

VAR_OUTPUT
	STATE_Last_Quartz:		INT;		(*dernier quartz utilisé*)
	STATE_Next_Quartz:		INT;		(*prochain quartz prévu*)
	OUT_Quartz:				INT;		(*quartz demandé en début de prod*)
	STATE_Mode:				BOOL;		(*mode 1run = 1quartz actif*)
	STATE_RAZ_Quartz:		BOOL;		(*le changement des quartz sera demandé au prochain run*)
	RQ_Disp_Change_Quartz:	BOOL;		(*affichage message "changement de tous les quartz pour le prochain run nécessaire*)
	RQ_Disp_Confirm_Quatz:	BOOL;		(*affichage demande confirmation de changement des quartz*)
	RQ_Pos_Quartz:			BOOL;		(*demande positionnement du quartz si quartz prévu en défaut*)
END_VAR

VAR
	RCP_M_Mode:				BOOL;
	RCP_M_RAZ_Quartz:		BOOL;
	VAR_Def_No_Quartz:		BOOL;
	FM_Mode:				R_TRIG;
	FM_Prod:				R_TRIG;
	FM_CD6T:				R_TRIG;
END_VAR

VAR_INPUT PERSISTENT
	CONF_N_Quartz_total:	INT;		(*nombre de quartz de la tete*)
	CONF_N_Quartz_secours:	INT;		(*nombre de quartz de secours à conserver avant de changer*)
	
	(*Entité*)
	IsFunction:		BOOL;			(*entité : assembly*)
	IdXML:			STRING;			(*nom entité : identifiant pour recherche dans dico*)
	TagXML:			UINT;			(*nom entité : identifiant pour recherche dans dico*)
	IdParent:		STRING;			(*MNEMO de l'appelant*)
	MNEMO:			STRING;			(*MNEMO de l'entité*)
END_VAR

(*réception des demandes*)
RCP_M_Mode			:=	M_Mode;
RCP_M_RAZ_Quartz	:=	M_RAZ_Quartz;

(*Changement de mode*)
IF STATE_Mode AND RCP_M_Mode AND NOT I_Prod THEN
	STATE_Mode	:=	FALSE;
ELSIF NOT STATE_Mode AND RCP_M_Mode AND NOT I_Prod THEN
	STATE_Mode	:=	TRUE;
END_IF

(*Forcage changement des quartz*)
FM_Mode(CLK := STATE_Mode);
IF STATE_RAZ_Quartz AND RCP_M_RAZ_Quartz THEN
	STATE_RAZ_Quartz	:=	FALSE;
ELSIF NOT STATE_RAZ_Quartz AND RCP_M_RAZ_Quartz THEN
	STATE_RAZ_Quartz	:=	TRUE;
END_IF

(*Gestion mémoire denier quartz utilisé*)
IF I_Prod AND I_Evap AND STATE_Mode THEN
	STATE_Last_Quartz	:=	I_Current_Quartz;
ELSIF FM_Mode.Q THEN
	STATE_Last_quartz	:=	0;
END_IF

(*Gestion prochain quartz affiché*)
IF (STATE_Last_Quartz >= (CONF_N_Quartz_total - CONF_N_Quartz_secours)) 
	OR (STATE_Last_quartz = 0) OR STATE_RAZ_Quartz THEN
		STATE_Next_Quartz	:=	1;
ELSE
		STATE_Next_Quartz	:=	STATE_Last_quartz + 1;
END_IF
idxml	:=	'21';
tagxml	:=	1;

(*Gestion quartz de consigne en début de procédé*)
FM_Prod(CLK := I_Prod);
IF FM_Prod.Q AND STATE_Mode THEN
	IF(STATE_Last_Quartz >= (CONF_N_Quartz_total - CONF_N_Quartz_secours)) 
		OR (STATE_Last_quartz = 0) OR STATE_RAZ_Quartz THEN
			OUT_Quartz			:=	1;
			STATE_RAZ_Quartz	:=	FALSE;
	ELSE
			OUT_Quartz			:=	STATE_Last_quartz + 1;
	END_IF
	WHILE I_QF[OUT_Quartz] AND (OUT_Quartz <= (CONF_N_Quartz_total - CONF_N_Quartz_secours)) DO
		OUT_Quartz	:=	OUT_Quartz + 1;
	END_WHILE
	IF I_QF[OUT_Quartz] OR  (OUT_Quartz > (CONF_N_Quartz_total - CONF_N_Quartz_secours)) THEN
		VAR_Def_No_Quartz	:=	TRUE;
	ELSE
		RQ_Pos_Quartz		:=	TRUE;
		STATE_Next_Quartz	:=	OUT_Quartz;
	END_IF
ELSE
	RQ_Pos_Quartz	:=	FALSE;
END_IF

(*Affichage demande confirmation changement quartz dans launcher*)
RQ_Disp_Confirm_Quatz	:=	(STATE_Next_Quartz = 1) AND NOT I_Prod AND STATE_Mode;

(*Affichage changement tous les quartz au prochain run*)
RQ_Disp_Change_Quartz	:=	(STATE_Next_Quartz = 1) AND STATE_Mode;

(*Défaut switch quartz trop nombreux*)
FM_CD6T(CLK := I_CD6T);
DEF_Stop_Quartz(
	IdXML		:=	'14',
	tagxml		:=	29,
	CONDITION 	:= 	FM_CD6T.Q AND I_Evap AND (I_Current_Quartz >= OUT_Quartz + CONF_N_Quartz_secours) AND STATE_Mode,
	DELAY		:=	T#0MS,
	);
	
(*Défaut pas de quartz pour la production*)
IF NOT I_Prod THEN
	VAR_Def_No_Quartz	:=	FALSE;
END_IF
DEF_No_Quartz(
	IdXML		:=	'14',
	tagxml		:=	30,
	CONDITION 	:= 	VAR_Def_No_Quartz,
	DELAY		:=	T#0MS,
	);

(*Reset des demandes*)
M_Mode					:=	FALSE;
M_RAZ_Quartz			:=	FALSE;

END_FUNCTION_BLOCK

// ---- POUs/FONCTION DE BASE/BLOCK_USER.TcPOU
FUNCTION_BLOCK BLOCK_USER
(* --------------------------------------------------------------------------------------- *)
(* Fonction de gestion des utilisateurs                                               *)
(* Gestion jusqu'à 10 groupes d'utilisateurs et 20 utilisateurs     *)
(* Version 0 - SP - 02/2012 - 7326 BA8						*)
(* Version 0.1 - AB - rebouclage droit demodif en ligne sur droit                            *)
(* ---------------------------------------------------------------------------------------  *)

VAR
	PREVIOUS_USER:	STRING;		(*nom du dernier utilisateur*)
	CONNECTED_USER:		STRING;		(*nom de l'actuel utilisateur*)
	{attribute 'OPC.UA.DA' := '1'}
	ACTU_USER:		USER_ACTU;
	USER_TEMP:		USER;
	GROUP_TEMP:		USER_GROUP;
	MANUFACTURER:	BOOL;	(*Indique que le fabriquant de la machine est connecté*)

	LOAD_EC:			BOOL;
	SAVE_EC:			BOOL;
	STOP_GROUP:		BOOL;
	STOP_USER:		BOOL;

	LOG_TEMP:			STRING[30];
	PASS_TEMP:			STRING[30];
	PASS_TEMP_DISPLAY:	STRING[30];

	UTIL_EC:			BOOL;
	LOG_EC:				STRING[30];
	INIT_DROIT:			BOOL;

	DD_LOG1:			BOOL;				(* Init avant page log *)
	DD_LOG:			BOOL;				(* Demande de connexion *)
	DD_DELOG:			BOOL;				(* Demande de déconnexion *)
	DD_NEW_USER:		BOOL;				(* Demande de création nouvelle utilisateur *)
	DD_NEW_GROUP:	BOOL;				(* Demande de création nouveau groupe *)
	DD_EFFACE_NEW:	BOOL;				(* Demande init avant page création user *)
	DD_EFFACE_NEW2:	BOOL;				(* Demande init avant page création groupe *)
	DD_DEL_USER:		BOOL;				(* Demande de suppression utilisateur *)
	DD_DEL_GROUP:	BOOL;				(* Demande de suppression groupe *)
	DD_mod_group1:		BOOL;				(* Demande inut avant page modification groupe *)
	DD_mod_group2:		BOOL;				(* Demande de modification d'un groupe *)
	DD_mod_user1:		BOOL;				(* Demande inut avant page modification user *)
	DD_mod_user2:		BOOL;				(* Demande de modification d'un user *)
	DD_sauv:			BOOL;				(* Demande de sauvegarde de la liste utilisateurs *)
	DD_load:			BOOL;				(* Demande de chargement liste utilisateurs *)
	DD_mod_def1:		BOOL;				(* Demande init avant page modification droits par défaut *)
	DD_mod_def2:		BOOL;				(* Demande modification droits par défaut *)
	DD_ORG_GRP:		BOOL;				(* Demande organisation groupe *)
	DD_ORG_USER:		BOOL;				(* Demande organisation utilisateur *)

	UTIL_INEXISTANT:	BOOL;				(* Utilisateur non trouvé *)
	GROUP_INEXISTANT:	BOOL;				(* Groupe non trouvé *)
	UTIL_EXIST:			BOOL;				(* Utilisateur deja existant *)
	GROUP_EXIST:		BOOL;				(* Groupe deja existant *)
	DEL_GROUP_IMPOS:	BOOL;				(* Suppression groupe impossible *)

	FCT_Ouv_File:		FB_FileOpen;			(*Fonction d'ouverture du fichier*)
	FCT_Write_File:		FB_FileWrite;
	FCT_Ferm_File:		FB_FileClose;
	FCT_Read_File:		FB_FileGets;

	hDestFile:			UINT	:= 0;
	Buffer:				STRING[30];
	Buff2:				STRING;
	NB:					INT;
	NB2:				INT;
	TROUV:				BOOL;
	TROUV2:			BOOL;
	LIGNE:				INT:=1;
	LIGNE_GROUP:		INT:=1;
	ITER:				INT;
	ITER2:				INT;
	ITER3:				INT;
	ITER4:				INT;
	Step:				INT;
	Step2:				INT;
	cbReadLength: 		UDINT;

	Patch_file:			STRING;

	AUT_MOD_GRP:		BOOL;					(* Autorisation modification et suppression groupe *)
	AUT_NOM_GRP:		BOOL;					(* Autorisation nom du groupe *)
	AUT_MOD_USER:	BOOL;					(* Autorisation modification et suppression utilisateur *)
	AUT_NOM_USER:	BOOL;					(* Autorisation nom de l'utilisateur *)
	AUT_NEW_USER:	BOOL;					(* Autorisation création utlisateur *)
	AUT_OPT_LOGOUT:	BOOL;					(* Autorisation utilisation logout auto *)

	NB_GROUP:		INT;
	NB_USER:		INT;

	TPS_ECOUL:		TON;						(* Temps écoulé pour le logout auto *)

	VISU_FEN1:		BOOL;
	VISU_FEN2:		BOOL;
	VISU_FEN3:		BOOL;
	VISU_FEN4:		BOOL;

	PASS_CONF:			STRING[30];
	PASS_CONF_DISPLAY:	STRING[30];
	FM_UTIL_EC:		R_TRIG;
	FD_UTIL_EC:		F_TRIG;
END_VAR

VAR_INPUT
	EV_CONNECT:		PRCDEF;	(*evenement de connexion d'un nouvel utilisateur*)
	EV_DISCONNECT:	PRCDEF;	(*evenement de déconnexion d'un nouvel utilisateur*)
END_VAR

VAR PERSISTENT
	OPT_LOGOUT:			BOOL;
	TIM_LOGOUT:			TIME;
	TBL_USER:				ARRAY [0..501] OF USER;
	TBL_GROUP:			ARRAY [0..50] OF USER_GROUP;
	GROUP_DEFAUT:		USER_GROUP;
	(* Entité*)
	IsFunction:		BOOL;			(*entité : ensemble*)
	IdXML:			STRING;			(*nom entité : identifiant pour recherche dans dico*)
	TagXML:			UINT;			(*nom entité : identifiant pour recherche dans dico*)
	IdParent:			STRING;			(*MNEMO de l'appelant*)
	MNEMO:			STRING;			(*MNEMO de l'entité*)
END_VAR

IF NOT PARAM_SYSTEM_OK THEN
	IdParent	:= MACHINE.MNEMO ;
	IdXML:='14';
	TagXML:=1;
	EV_CONNECT.Groupe :=2;
	EV_DISCONNECT.Groupe :=2;
	EV_CONNECT.IdXML := '15';
	EV_DISCONNECT.IdXML := '15';
	EV_CONNECT.tagXML := 1;
	EV_DISCONNECT.tagXML := 2;
	MNEMO:='USER';
END_IF

(*affichage codé des password*)
IF USER_TEMP.PASS <> '' THEN
	USER_TEMP.PASS_DISPLAY := '*****';
ELSE
	USER_TEMP.PASS_DISPLAY := '';	
END_IF

IF PASS_TEMP <> '' THEN
	PASS_TEMP_DISPLAY := '*****';
ELSE
	PASS_TEMP_DISPLAY := '';
END_IF

IF PASS_CONF <> '' THEN
	PASS_CONF_DISPLAY := '*****';
ELSE
	PASS_CONF_DISPLAY := '';
END_IF



IF LIGNE < 1 THEN
	LIGNE := 1;
END_IF
IF LIGNE_GROUP < 1 THEN
	LIGNE_GROUP := 1;	
END_IF

(* Error Code :
01 / L"utilisateur n"existe pas ou le mot de passe n"est pas bon
02 / Le groupe utilisateur n"est plus présent.
03 / Veuillez sélectionner un groupe valide.  
04 / Un autre utilisateur possède le meme identifiant. 
05 / Ce groupe existe déjà !
06 / Un utilisateur possède ce groupe. Suppression impossible
07 / Le fichier de sauvegarde n"est pas accessible.
08 / Erreur d"écriture dans le fichier.
09 / Erreur de fermeture du fichier.
10 / Le fichier de sauvegarde n"est pas accessible.
11 / Problème de lecture du fichier.
12 / Erreur de fermeture du fichier. *)

Patch_file		:=	'C:\Machine\User\Sauv.util';

NB_GROUP	:=	10;		(* Max 50 *)
NB_USER		:=	500;		(* Max 100 *)

(*************************************** Initialisation des droits utilisateurs **********************************************)
(* si pas d'utilisateur connecté, on applique les droits par défaut									    *)

IF NOT UTIL_EC THEN
	ACTU_USER.GROUPE				:=	'Default';
	ACTU_USER.CONF_MACHINE			:=	GROUP_DEFAUT.CONF_MACHINE;
	ACTU_USER.FONCTION_SA			:=	GROUP_DEFAUT.FONCTION_SA;
	ACTU_USER.MAINTENANCE			:=	GROUP_DEFAUT.MAINTENANCE;
	ACTU_USER.PRODUCTION			:=	GROUP_DEFAUT.PRODUCTION;
	ACTU_USER.PROGRAMMATION			:=	GROUP_DEFAUT.PROGRAMMATION;
	ACTU_USER.SUPERVISEUR			:=	GROUP_DEFAUT.SUPERVISEUR;
	ACTU_USER.CONF_TRF				:=	GROUP_DEFAUT.CONF_TRF;
	ACTU_USER.MODIF_ENLIGNE			:=	GROUP_DEFAUT.MODIF_ENLIGNE OR GROUP_DEFAUT.PROGRAMMATION;
	ACTU_USER.ARCHIVE_EV			:=	GROUP_DEFAUT.ARCHIVE_EV;
	ACTU_USER.DECONSIGNATION		:=	GROUP_DEFAUT.DECONSIGNATION;
END_IF
(*=======================================================================================*)


(************************************************* Demande de déconnexion *********************************************)
IF DD_DELOG THEN
	IF UTIL_EC THEN
			IF NOT (ACTU_USER.PRENOM  = '') OR NOT (ACTU_USER.NOM = '') THEN
				PREVIOUS_USER:=CONCAT(ACTU_USER.PRENOM, CONCAT(' ',ACTU_USER.NOM));
			ELSE
				PREVIOUS_USER:=ACTU_USER.LOGIN;
			END_IF
	END_IF
	CONNECTED_USER := '';
	ACTU_USER.GROUPE			:=	'';
	ACTU_USER.LOGIN				:=	'';
	ACTU_USER.NOM				:=	'';
	ACTU_USER.PASS				:=	'';
	ACTU_USER.PRENOM			:=	'';
	ACTU_USER.CONF_MACHINE		:=	FALSE;
	ACTU_USER.FONCTION_SA		:=	FALSE;
	ACTU_USER.MAINTENANCE		:=	FALSE;
	ACTU_USER.PRODUCTION		:=	FALSE;
	ACTU_USER.PROGRAMMATION		:=	FALSE;
	ACTU_USER.SUPERVISEUR		:=	FALSE;
	ACTU_USER.CONF_TRF			:=	FALSE;
	ACTU_USER.MODIF_ENLIGNE		:=	FALSE;
	ACTU_USER.ARCHIVE_EV		:=	FALSE;
	ACTU_USER.DECONSIGNATION	:=	FALSE;
	UTIL_EC						:=	FALSE;
	DD_DELOG					:=	FALSE;
	MANUFACTURER				:=	FALSE;
END_IF
(*===================================================================================================*)


(************************************************* Demande d'ouverture  *********************************************)
(*									de la fenêtre de mot de passe						       *)
IF DD_LOG1 THEN
	LOG_TEMP 		:=	'';
	PASS_TEMP 	:=	'';
	DD_LOG1 		:=	FALSE;
END_IF
(*===================================================================================================*)

(************************************************* Demande de connexion *********************************************)
IF DD_LOG THEN

	TROUV	:=	FALSE;
	TROUV2	:=	FALSE;
	NB		:=	1;
	NB2		:=	1;

	IF	LOG_TEMP = 'ac' AND PASS_TEMP = 'ac' THEN
		ACTU_USER.LOGIN		:=	'Alliance-concept';
		ACTU_USER.CONF_MACHINE		:=	TRUE;
		ACTU_USER.FONCTION_SA		:=	TRUE;
		ACTU_USER.MAINTENANCE		:=	TRUE;
		ACTU_USER.PRODUCTION		:=	TRUE;
		ACTU_USER.PROGRAMMATION		:=	TRUE;
		ACTU_USER.SUPERVISEUR		:=	TRUE;
		ACTU_USER.CONF_TRF			:=	TRUE;
		ACTU_USER.MODIF_ENLIGNE		:=	TRUE;
		ACTU_USER.ARCHIVE_EV		:=	TRUE;
		ACTU_USER.DECONSIGNATION	:=	TRUE;
		ACTU_USER.GROUPE			:=	'';
		MANUFACTURER				:=	TRUE;
		UTIL_EC						:=	TRUE;
		CONNECTED_USER				:= 'Alliance Concept';
	ELSE
	MANUFACTURER:=FALSE;
	(*recherche de l'utilisateur dans la table des utilisateurs*)
		FOR NB := 1 TO NB_USER DO
			IF TBL_USER[NB].LOGIN	=	LOG_TEMP AND TBL_USER[NB].PASS	=	PASS_TEMP THEN
				TROUV	:=	TRUE;
				ACTU_USER.GROUPE	:=	TBL_USER[NB].GROUPE;
				ACTU_USER.LOGIN		:=	LOG_TEMP;
				ACTU_USER.NOM		:=	TBL_USER[NB].NOM;
				ACTU_USER.PASS		:=	TBL_USER[NB].PASS;
				ACTU_USER.PRENOM	:=	TBL_USER[NB].PRENOM;
			END_IF

			IF TROUV THEN

				FOR NB2 := 1 TO NB_GROUP DO
					IF TBL_GROUP[NB2].NOM	=	ACTU_USER.GROUPE THEN
						TROUV2		:=	TRUE;
						ACTU_USER.CONF_MACHINE		:=	TBL_GROUP[NB2].CONF_MACHINE;
						ACTU_USER.FONCTION_SA		:=	TBL_GROUP[NB2].FONCTION_SA;
						ACTU_USER.MAINTENANCE		:=	TBL_GROUP[NB2].MAINTENANCE;
						ACTU_USER.PRODUCTION		:=	TBL_GROUP[NB2].PRODUCTION;
						ACTU_USER.PROGRAMMATION	:=	TBL_GROUP[NB2].PROGRAMMATION;
						ACTU_USER.SUPERVISEUR		:=	TBL_GROUP[NB2].SUPERVISEUR;
						ACTU_USER.CONF_TRF			:=	TBL_GROUP[NB2].CONF_TRF;
						ACTU_USER.MODIF_ENLIGNE		:=	TBL_GROUP[NB2].MODIF_ENLIGNE OR TBL_GROUP[NB2].PROGRAMMATION;
						ACTU_USER.ARCHIVE_EV		:=	TBL_GROUP[NB2].ARCHIVE_EV;
						ACTU_USER.DECONSIGNATION	:=	TBL_GROUP[NB2].DECONSIGNATION;	(*droit modifié en maintenance non sécurisée*)
						IF NOT (ACTU_USER.PRENOM  = '') OR NOT (ACTU_USER.NOM = '') THEN
							CONNECTED_USER:=CONCAT(ACTU_USER.PRENOM, CONCAT(' ',ACTU_USER.NOM));
						ELSE
							CONNECTED_USER:=ACTU_USER.LOGIN;
						END_IF
						UTIL_EC							:=	TRUE;
					END_IF;
				END_FOR;
			END_IF
		END_FOR;

	END_IF
(*
	IF NOT TROUV AND NB >= NB_USER THEN
			(* Rajout controle code débloquage *)
			IF LEN(LOG_TEMP) = 8  AND LEN(PASS_TEMP) = 8 THEN
				PRG_SEC.Id_tp			:=	LOG_TEMP;
				PRG_SEC.Mdp_tp		:=	PASS_TEMP;
				PRG_SEC.DD_Deblok	:=	TRUE;
				TROUV2				:=	TRUE;
			ELSE
				ADSLOGSTR( msgCtrlMask := ADSLOG_MSGTYPE_ERROR OR ADSLOG_MSGTYPE_MSGBOX,
	        				msgFmtStr :=  'Error Code 1', strArg := ''); (* L"utilisateur n"existe pas ou le mot de passe n"est pas bon. *)
			END_IF
	END_IF
*)
	IF NOT TROUV2 AND NB2 >= NB_GROUP THEN
		ADSLOGSTR( msgCtrlMask := ADSLOG_MSGTYPE_ERROR OR ADSLOG_MSGTYPE_MSGBOX,
        				msgFmtStr :=  'Error Code 2', strArg := ''); (* Le groupe utilisateur n"est plus présent. *)
	END_IF

	DD_LOG	:=	FALSE;
END_IF
(*Gestion des événements de connexion*)
FM_UTIL_EC(CLK:=UTIL_EC);
FD_UTIL_EC(CLK:=UTIL_EC);
EV_CONNECT(
	CONDITION:=FM_UTIL_EC.Q ,
	VAL1:= CONNECTED_USER
	);
EV_DISCONNECT(
	CONDITION:=FD_UTIL_EC.Q ,
	VAL1:= PREVIOUS_USER

	);

(*===================================================================================================*)


(************************************************* Demande de création d'un nouvel utilisateur *********************************************)
IF DD_NEW_USER THEN
	NB2		:=	0;

	IF TBL_GROUP[LIGNE_GROUP].NOM = '' THEN
			ADSLOGSTR( msgCtrlMask := ADSLOG_MSGTYPE_ERROR OR ADSLOG_MSGTYPE_MSGBOX,
        				msgFmtStr :=  'Error Code 3', strArg := ''); (* Veuillez sélectionner un groupe valide. *)
		GROUP_INEXISTANT	:=	TRUE;
	END_IF

	IF USER_TEMP.LOGIN <> '' AND USER_TEMP.LOGIN <> ' ' AND NOT GROUP_INEXISTANT THEN

		FOR NB := 1 TO NB_USER DO

			IF TBL_USER[NB].LOGIN	=	USER_TEMP.LOGIN THEN
				UTIL_EXIST	:=	TRUE;
			END_IF

			IF TBL_USER[NB].LOGIN = '' AND NB2	= 0 THEN
				NB2	:=	NB;
			END_IF

		END_FOR

	END_IF

	IF UTIL_EXIST THEN
		ADSLOGSTR( msgCtrlMask := ADSLOG_MSGTYPE_ERROR OR ADSLOG_MSGTYPE_MSGBOX,
			msgFmtStr :=  'Error Code 4', strArg := ''); (* Un autre utilisateur possède le meme identifiant. *)
	END_IF

	IF UTIL_EXIST = FALSE AND NB2 > 0 AND NOT GROUP_INEXISTANT THEN
		TBL_USER[NB2].LOGIN		:=	USER_TEMP.LOGIN;
		TBL_USER[NB2].NOM			:=	USER_TEMP.NOM;
		TBL_USER[NB2].PRENOM		:=	USER_TEMP.PRENOM;
		TBL_USER[NB2].PASS		:=	USER_TEMP.PASS;
		TBL_USER[NB2].GROUPE		:=	TBL_GROUP[LIGNE_GROUP].NOM;
	END_IF

	DD_NEW_USER	:=	FALSE;			(*RAZ de la demande*)
	RQ_SAV_PERSISTENT := TRUE;		(*Demande de sauvegarde des variables*)

ELSE
	GROUP_INEXISTANT	:=	FALSE;
	UTIL_EXIST			:=	FALSE;
END_IF
(*===================================================================================================*)


(************************************************* Chargement page nouvelle utilisateur *********************************************)
IF DD_EFFACE_NEW THEN
	USER_TEMP.GROUPE	:=	'';
	USER_TEMP.LOGIN		:=	'';
	USER_TEMP.NOM		:=	'';
	USER_TEMP.PASS		:=	'';
	USER_TEMP.PRENOM	:=	'';
	PASS_CONF			:=	'';
	DD_EFFACE_NEW		:=	FALSE;
END_IF
(*===================================================================================================*)


(************************************************* Demande de création d'un groupe *********************************************)
IF DD_NEW_GROUP THEN

	FOR NB := 1 TO NB_GROUP DO
		IF TBL_GROUP[NB].NOM = GROUP_TEMP.NOM THEN
			GROUP_EXIST := TRUE;
				ADSLOGSTR( msgCtrlMask := ADSLOG_MSGTYPE_ERROR OR ADSLOG_MSGTYPE_MSGBOX,
        				msgFmtStr :=  'Error Code 5', strArg := ''); (* Ce groupe existe déjà ! *)
		END_IF
	END_FOR

	IF NOT GROUP_EXIST THEN
		NB2		:=	0;
		FOR NB := 1 TO NB_GROUP DO
			IF TBL_GROUP[NB].NOM = '' AND NB2 = 0 THEN
				NB2		:=	NB;
			END_IF
		END_FOR
		IF NB2 > 0 THEN
			TBL_GROUP[NB2].NOM				:=	GROUP_TEMP.NOM;
			TBL_GROUP[NB2].CONF_MACHINE		:=	GROUP_TEMP.CONF_MACHINE;
			TBL_GROUP[NB2].FONCTION_SA		:=	GROUP_TEMP.FONCTION_SA;
			TBL_GROUP[NB2].MAINTENANCE		:=	GROUP_TEMP.MAINTENANCE;
			TBL_GROUP[NB2].PRODUCTION		:=	GROUP_TEMP.PRODUCTION;
			TBL_GROUP[NB2].PROGRAMMATION	:=	GROUP_TEMP.PROGRAMMATION;
			TBL_GROUP[NB2].SUPERVISEUR		:=	GROUP_TEMP.SUPERVISEUR;
			TBL_GROUP[NB2].CONF_TRF			:=	GROUP_TEMP.CONF_TRF;
			TBL_GROUP[NB2].MODIF_ENLIGNE	:=	GROUP_TEMP.MODIF_ENLIGNE;
			TBL_GROUP[NB2].ARCHIVE_EV		:=	GROUP_TEMP.ARCHIVE_EV;
			TBL_GROUP[NB2].DECONSIGNATION	:=	GROUP_TEMP.DECONSIGNATION;
		END_IF
	END_IF

	DD_NEW_GROUP	:=	FALSE;
	RQ_SAV_PERSISTENT	:=	TRUE;			(*Demande de sauvegarde des variables persistentes*)
ELSE
	GROUP_EXIST := FALSE;
END_IF
(*===================================================================================================*)


(************************************************* Chargement page nouveau groupe *********************************************)
IF DD_EFFACE_NEW2 THEN
	GROUP_TEMP.NOM		:=	'';
	GROUP_TEMP.CONF_MACHINE		:=	FALSE;
	GROUP_TEMP.FONCTION_SA			:=	FALSE;
	GROUP_TEMP.MAINTENANCE			:=	FALSE;
	GROUP_TEMP.PRODUCTION			:=	FALSE;
	GROUP_TEMP.PROGRAMMATION		:=	FALSE;
	GROUP_TEMP.SUPERVISEUR			:=	FALSE;
	GROUP_TEMP.CONF_TRF			:=	FALSE;
	GROUP_TEMP.MODIF_ENLIGNE		:=	FALSE;
	GROUP_TEMP.ARCHIVE_EV			:=	FALSE;
	GROUP_TEMP.DECONSIGNATION		:=	FALSE;
	DD_EFFACE_NEW2					:=	FALSE;
END_IF
(*===================================================================================================*)


(************************************************* Suppression d'un utilisateur *********************************************)
IF DD_DEL_USER THEN
	IF LIGNE > 0 THEN
		TBL_USER[LIGNE].NOM			:=	'';
		TBL_USER[LIGNE].GROUPE		:=	'';
		TBL_USER[LIGNE].LOGIN			:=	'';
		TBL_USER[LIGNE].PASS			:=	'';
		TBL_USER[LIGNE].PRENOM		:=	'';
	END_IF
	DD_DEL_USER	:=	FALSE;
	RQ_SAV_PERSISTENT	:= TRUE;
	DD_ORG_USER		:=	TRUE;
END_IF
(*===================================================================================================*)



(************************************************* Suppression d'un groupe *********************************************)
IF DD_DEL_GROUP THEN

	IF LIGNE_GROUP > 0 THEN
		FOR NB := 1 TO NB_USER DO
			IF TBL_USER[NB].GROUPE = TBL_GROUP[LIGNE_GROUP].NOM THEN
				ADSLOGSTR( msgCtrlMask := ADSLOG_MSGTYPE_ERROR OR ADSLOG_MSGTYPE_MSGBOX,
        				msgFmtStr :=  'Error Code 6', strArg := ''); (* Un utilisateur possède ce groupe. Suppression impossible *)
				DEL_GROUP_IMPOS	:=	TRUE;
			END_IF
		END_FOR
		IF NOT DEL_GROUP_IMPOS THEN
			TBL_GROUP[LIGNE_GROUP].NOM					:=	'';
			TBL_GROUP[LIGNE_GROUP].CONF_MACHINE		:=	FALSE;
			TBL_GROUP[LIGNE_GROUP].FONCTION_SA		:=	FALSE;
			TBL_GROUP[LIGNE_GROUP].MAINTENANCE		:=	FALSE;
			TBL_GROUP[LIGNE_GROUP].PRODUCTION			:=	FALSE;
			TBL_GROUP[LIGNE_GROUP].PROGRAMMATION	:=	FALSE;
			TBL_GROUP[LIGNE_GROUP].SUPERVISEUR		:=	FALSE;
			TBL_GROUP[LIGNE_GROUP].CONF_TRF			:=	FALSE;
			TBL_GROUP[LIGNE_GROUP].MODIF_ENLIGNE		:=	FALSE;
			TBL_GROUP[LIGNE_GROUP].ARCHIVE_EV			:=	FALSE;
			TBL_GROUP[LIGNE_GROUP].DECONSIGNATION	:=	FALSE;
		END_IF
	END_IF
	DD_DEL_GROUP	:=	FALSE;
	RQ_SAV_PERSISTENT := TRUE;
	DD_ORG_GRP			:=	TRUE;
ELSE
	DEL_GROUP_IMPOS		:=	FALSE;
END_IF
(*===================================================================================================*)



(************************************************* Init avant ouverture page modification groupe *********************************************)
IF DD_mod_group1 THEN
	GROUP_TEMP.CONF_MACHINE		:=	TBL_GROUP[LIGNE_GROUP].CONF_MACHINE;
	GROUP_TEMP.FONCTION_SA			:=	TBL_GROUP[LIGNE_GROUP].FONCTION_SA;
	GROUP_TEMP.MAINTENANCE			:=	TBL_GROUP[LIGNE_GROUP].MAINTENANCE;
	GROUP_TEMP.NOM					:=	TBL_GROUP[LIGNE_GROUP].NOM;
	GROUP_TEMP.PRODUCTION			:=	TBL_GROUP[LIGNE_GROUP].PRODUCTION;
	GROUP_TEMP.PROGRAMMATION		:=	TBL_GROUP[LIGNE_GROUP].PROGRAMMATION;
	GROUP_TEMP.SUPERVISEUR			:=	TBL_GROUP[LIGNE_GROUP].SUPERVISEUR;
	GROUP_TEMP.CONF_TRF			:=	TBL_GROUP[LIGNE_GROUP].CONF_TRF;
	GROUP_TEMP.MODIF_ENLIGNE		:=	TBL_GROUP[LIGNE_GROUP].MODIF_ENLIGNE;
	GROUP_TEMP.ARCHIVE_EV			:=	TBL_GROUP[LIGNE_GROUP].ARCHIVE_EV;
	GROUP_TEMP.DECONSIGNATION		:=	TBL_GROUP[LIGNE_GROUP].DECONSIGNATION;
	DD_mod_group1	:=	FALSE;
END_IF
(*===================================================================================================*)


(************************************************* Modification d'un groupe *********************************************)
IF DD_mod_group2 THEN
	TBL_GROUP[LIGNE_GROUP].CONF_MACHINE		:=	GROUP_TEMP.CONF_MACHINE;
	TBL_GROUP[LIGNE_GROUP].FONCTION_SA		:=	GROUP_TEMP.FONCTION_SA;
	TBL_GROUP[LIGNE_GROUP].MAINTENANCE		:=	GROUP_TEMP.MAINTENANCE;
	TBL_GROUP[LIGNE_GROUP].NOM					:=	GROUP_TEMP.NOM;
	TBL_GROUP[LIGNE_GROUP].PRODUCTION			:=	GROUP_TEMP.PRODUCTION;
	TBL_GROUP[LIGNE_GROUP].PROGRAMMATION	:=	GROUP_TEMP.PROGRAMMATION;
	TBL_GROUP[LIGNE_GROUP].SUPERVISEUR		:=	GROUP_TEMP.SUPERVISEUR	;
	TBL_GROUP[LIGNE_GROUP].CONF_TRF			:=	GROUP_TEMP.CONF_TRF;
	TBL_GROUP[LIGNE_GROUP].MODIF_ENLIGNE		:=	GROUP_TEMP.MODIF_ENLIGNE;
	TBL_GROUP[LIGNE_GROUP].ARCHIVE_EV			:=	GROUP_TEMP.ARCHIVE_EV;
	TBL_GROUP[LIGNE_GROUP].DECONSIGNATION	:=	GROUP_TEMP.DECONSIGNATION;
	DD_mod_group2	:=	FALSE;
	RQ_SAV_PERSISTENT	:= TRUE;		(*Ecriture des variables persitante*)
END_IF
(*===================================================================================================*)



(************************************************* Init avant ouverture page modification groupe defaut *********************************************)
IF DD_mod_def1 THEN
	GROUP_TEMP.CONF_MACHINE		:=	GROUP_DEFAUT.CONF_MACHINE;
	GROUP_TEMP.FONCTION_SA			:=	GROUP_DEFAUT.FONCTION_SA;
	GROUP_TEMP.MAINTENANCE			:=	GROUP_DEFAUT.MAINTENANCE;
	GROUP_TEMP.PRODUCTION			:=	GROUP_DEFAUT.PRODUCTION;
	GROUP_TEMP.PROGRAMMATION		:=	GROUP_DEFAUT.PROGRAMMATION;
	GROUP_TEMP.SUPERVISEUR			:=	GROUP_DEFAUT.SUPERVISEUR;
	GROUP_TEMP.CONF_TRF			:=	GROUP_DEFAUT.CONF_TRF;
	GROUP_TEMP.MODIF_ENLIGNE		:=	GROUP_DEFAUT.MODIF_ENLIGNE;
	GROUP_TEMP.ARCHIVE_EV			:=	GROUP_DEFAUT.ARCHIVE_EV;
	GROUP_TEMP.DECONSIGNATION		:=	GROUP_DEFAUT.DECONSIGNATION;
	 DD_mod_def1	:=	FALSE;
END_IF
(*===================================================================================================*)

(************************************************* Demande modification des droits par défaut  *********************************************)
IF DD_mod_def2 THEN
	GROUP_DEFAUT.CONF_MACHINE		:=	GROUP_TEMP.CONF_MACHINE;
	GROUP_DEFAUT.FONCTION_SA		:=	GROUP_TEMP.FONCTION_SA;
	GROUP_DEFAUT.MAINTENANCE		:=	GROUP_TEMP.MAINTENANCE;
	GROUP_DEFAUT.NOM				:=	'Default';
	GROUP_DEFAUT.PRODUCTION		:=	GROUP_TEMP.PRODUCTION;
	GROUP_DEFAUT.PROGRAMMATION	:=	GROUP_TEMP.PROGRAMMATION;
	GROUP_DEFAUT.SUPERVISEUR		:=	GROUP_TEMP.SUPERVISEUR;
	GROUP_DEFAUT.CONF_TRF			:=	GROUP_TEMP.CONF_TRF;
	GROUP_DEFAUT.MODIF_ENLIGNE		:=	GROUP_TEMP.MODIF_ENLIGNE;
	GROUP_DEFAUT.ARCHIVE_EV		:=	GROUP_TEMP.ARCHIVE_EV;
	GROUP_DEFAUT.DECONSIGNATION	:=	GROUP_TEMP.DECONSIGNATION;
	RQ_SAV_PERSISTENT				:= TRUE;		(*Ecriture des variables persistentes*)
	DD_mod_def2	:=	FALSE;
END_IF
(*===================================================================================================*)


(************************************************* Init avant ouverture page modification user *********************************************)
IF DD_mod_user1 THEN
	USER_TEMP.GROUPE		:=	TBL_USER[LIGNE].GROUPE;
	USER_TEMP.LOGIN			:=	TBL_USER[LIGNE].LOGIN;
	USER_TEMP.NOM			:=	TBL_USER[LIGNE].NOM;
	USER_TEMP.PASS			:=	TBL_USER[LIGNE].PASS;
	USER_TEMP.PRENOM		:=	TBL_USER[LIGNE].PRENOM;
	DD_mod_user1	:=	FALSE;
END_IF
(*===================================================================================================*)


(************************************************* Modification d'un user *********************************************)
IF DD_mod_user2 THEN
	TBL_USER[LIGNE].GROUPE		:=		TBL_GROUP[LIGNE_GROUP].NOM;
	TBL_USER[LIGNE].LOGIN			:=		USER_TEMP.LOGIN;
	TBL_USER[LIGNE].NOM			:=		USER_TEMP.NOM;
	TBL_USER[LIGNE].PASS			:=		USER_TEMP.PASS;
	TBL_USER[LIGNE].PRENOM		:=		USER_TEMP.PRENOM;
	DD_mod_user2	:=	FALSE;
	RQ_SAV_PERSISTENT 			:=	TRUE;	(*Ecriture des variables persistante*)
END_IF
(*===================================================================================================*)





(************************************************* Sauvegarde des utilisateurs *********************************************)
IF DD_sauv THEN
	Step	:=	1;
	DD_sauv	:=	FALSE;
END_IF

CASE Step OF
	0:(* do nothing *)
	ITER := 1;
	ITER2 := 1;

	1:
		(*OUVERTURE*)
		FCT_Ouv_File( bExecute := FALSE );
		FCT_Ouv_File(
			sNetId:=			'' ,
			sPathName := 	Patch_file,
			nMode:= 			FOPEN_MODEWRITE,
			ePath:= 			PATH_GENERIC,
			tTimeout:= 		T#10s,
			bExecute:=		TRUE
			 );
		Step := Step + 1;

	2:
		FCT_Ouv_File( bExecute := FALSE );
		IF ( NOT FCT_Ouv_File.bBusy ) THEN
			IF ( FCT_Ouv_File.bError ) THEN
				ADSLOGSTR( msgCtrlMask := ADSLOG_MSGTYPE_ERROR ,
	        			msgFmtStr :=  'Error Code 7', strArg := ''); (* Le fichier de sauvegarde n"est pas accessible. *)
				Step := 50;
			ELSE
				hDestFile := FCT_Ouv_File.hFile;
				Step := Step + 1;
			END_IF
		END_IF


	3:
		IF ITER2 <= NB_GROUP THEN
			CASE ITER OF
				1:
					Buffer	:=	CONCAT(TBL_GROUP[ITER2].NOM,'$N');
				2:
					Buffer	:=	CONCAT(BOOL_TO_STRING(TBL_GROUP[ITER2].CONF_MACHINE),'$N');
				3:
					Buffer	:=	CONCAT(BOOL_TO_STRING(TBL_GROUP[ITER2].FONCTION_SA),'$N');
				4:
					Buffer	:=	CONCAT(BOOL_TO_STRING(TBL_GROUP[ITER2].MAINTENANCE),'$N');
				5:
					Buffer	:=	CONCAT(BOOL_TO_STRING(TBL_GROUP[ITER2].PRODUCTION),'$N');
				6:
					Buffer	:=	CONCAT(BOOL_TO_STRING(TBL_GROUP[ITER2].PROGRAMMATION),'$N');
				7:
					Buffer	:=	CONCAT(BOOL_TO_STRING(TBL_GROUP[ITER2].SUPERVISEUR),'$N');
				8:
					Buffer	:=	CONCAT(BOOL_TO_STRING(TBL_GROUP[ITER2].CONF_TRF),'$N');
				9:
					Buffer	:=	CONCAT(BOOL_TO_STRING(TBL_GROUP[ITER2].MODIF_ENLIGNE),'$N');
				10:
					Buffer	:=	CONCAT(BOOL_TO_STRING(TBL_GROUP[ITER2].ARCHIVE_EV),'$N');
				11:
					Buffer	:=	CONCAT(BOOL_TO_STRING(TBL_GROUP[ITER2].DECONSIGNATION),'$N');
			END_CASE
		ELSE
			CASE ITER OF
				1:
					Buffer	:=	CONCAT(TBL_USER[ITER2-NB_GROUP].GROUPE,'$N');
				2:
					Buffer	:=	CONCAT(TBL_USER[ITER2-NB_GROUP].LOGIN,'$N');
				3:
					Buffer	:=	CONCAT(TBL_USER[ITER2-NB_GROUP].NOM,'$N');
				4:
					Buffer	:=	CONCAT(TBL_USER[ITER2-NB_GROUP].PASS,'$N');
				5:
					Buffer	:=	CONCAT(TBL_USER[ITER2-NB_GROUP].PRENOM,'$N');
			END_CASE
		END_IF

		FCT_Write_File( bExecute := FALSE );
		FCT_Write_File(sNetId:='',
				hFile:=hDestFile,
				pWriteBuff:= ADR(Buffer),
				cbWriteLen	:=	FIND(Buffer,'$N'),
				bExecute:=TRUE,
				tTimeout:=T#10s );
		Step := Step + 1;
		ITER	:=	ITER + 1;

	4:
		FCT_Write_File( bExecute := FALSE );
		IF ( NOT FCT_Write_File.bBusy ) THEN
			IF ( FCT_Write_File.bError ) THEN
				ADSLOGSTR( msgCtrlMask := ADSLOG_MSGTYPE_ERROR ,
    					msgFmtStr :=  'Error Code 8', strArg := '');	(* Erreur d"écriture dans le fichier. *)
				Step := 50;
			ELSE
				IF ITER > 11 AND ITER2 <= NB_GROUP THEN
					ITER2 := ITER2 + 1;
					ITER := 1;
				ELSE
					IF ITER > 5 AND ITER2 > NB_GROUP THEN
						ITER2 := ITER2 + 1;
						IF ITER2 > NB_GROUP + NB_USER THEN
							Step := 50;
						ELSE
							ITER := 1;
							Step := 3;
						END_IF
					ELSE
						Step := 3;
					END_IF
				END_IF
			END_IF
		END_IF

	30:
		FCT_Ferm_File( bExecute := FALSE );
		FCT_Ferm_File( 	sNetId:='',
				hFile:=hDestFile,
				bExecute:=TRUE,
				tTimeout:=T#10s  );
		Step := Step + 1;

	31:
		FCT_Ferm_File( bExecute := FALSE );
		IF ( NOT FCT_Ferm_File.bBusy ) THEN
			IF ( FCT_Ferm_File.bError ) THEN
				ADSLOGSTR( msgCtrlMask := ADSLOG_MSGTYPE_ERROR ,
        				msgFmtStr :=  'Error Code 9', strArg := '');	(* Erreur de fermeture du fichier. *)
			ELSE
				ADSLOGSTR( msgCtrlMask := ADSLOG_MSGTYPE_MSGBOX,
        				msgFmtStr :=  'OK !', strArg := '');
			END_IF
			Step := 50;
			hDestFile := 0;
		END_IF

	50:
		IF ( hDestFile <> 0 ) THEN
			Step := 30; (* close the destination file*)
		ELSE
			Step	:=	0;
		END_IF

END_CASE
(*===================================================================================================*)


(************************************************* Chargement des utilisateurs *********************************************)
IF DD_load THEN
	Step2	:=	1;
	DD_load	:=	FALSE;
	ITER3 := 1;
	ITER4 := 1;
END_IF

CASE Step2 OF
	0:(* do nothing *)
	;

	1:
		(*OUVERTURE*)
		FCT_Ouv_File( bExecute := FALSE );
		FCT_Ouv_File(
			sNetId:=			'' ,
			sPathName := 	Patch_file,
			nMode:= 			FOPEN_MODEREAD OR FOPEN_MODEBINARY,
			ePath:= 			PATH_GENERIC,
			tTimeout:= 		T#10s,
			bExecute:=		TRUE
			 );
		Step2 := Step2 + 1;

	2:
		FCT_Ouv_File( bExecute := FALSE );
		IF ( NOT FCT_Ouv_File.bBusy ) THEN
			IF ( FCT_Ouv_File.bError ) THEN
				ADSLOGSTR( msgCtrlMask := ADSLOG_MSGTYPE_ERROR ,
	        			msgFmtStr :=  'Error Code 10', strArg := ''); (* Le fichier de sauvegarde n"est pas accessible. *)
				Step2 := 50;
			ELSE
				hDestFile := FCT_Ouv_File.hFile;
				Step2 := Step2 + 1;
			END_IF
		END_IF

	3:
		FCT_Read_File( bExecute:= FALSE );
		FCT_Read_File( 	sNetId:='',
				hFile:=hDestFile,
				bExecute:=TRUE,
				tTimeout:=T#10s );
		Step2 := Step2 + 1;

	4:
		FCT_Read_File( bExecute:= FALSE );
		IF ( NOT FCT_Read_File.bBusy ) THEN
			IF ( FCT_Read_File.bError ) THEN
				ADSLOGSTR( msgCtrlMask := ADSLOG_MSGTYPE_ERROR ,
	        			msgFmtStr :=  'Error Code 11', strArg := ''); (* Problème de lecture du fichier. *)
				Step2 := 50;
			ELSE
				Buff2 := FCT_Read_File.sLine;
				IF FCT_Read_File.bEOF THEN
					Step2 := 50;
				ELSE
					Step2 := Step2 + 1;
				END_IF
			END_IF
		END_IF

	5:

		IF ITER4 <= NB_GROUP THEN
			IF ITER3 > 11 THEN
				ITER3 := 1;
				ITER4 := ITER4 + 1;
				IF ITER4 <= NB_GROUP THEN
					TBL_GROUP[ITER4].NOM	:=	MID(Buff2,FIND(Buff2,'$R')-1,1);
				ELSE
					TBL_USER[ITER4-NB_GROUP].GROUPE			:=	MID(Buff2,FIND(Buff2,'$R')-1,1);
				END_IF
			ELSE
				CASE ITER3 OF
					1:
						TBL_GROUP[ITER4].NOM	:=	MID(Buff2,FIND(Buff2,'$R')-1,1);
					2:
						TBL_GROUP[ITER4].CONF_MACHINE	:=	STRING_TO_BOOL(MID(Buff2,FIND(Buff2,'$R')-1,1));
					3:
						TBL_GROUP[ITER4].FONCTION_SA	:=	STRING_TO_BOOL(MID(Buff2,FIND(Buff2,'$R')-1,1));
					4:
						TBL_GROUP[ITER4].MAINTENANCE	:=	STRING_TO_BOOL(MID(Buff2,FIND(Buff2,'$R')-1,1));
					5:
						TBL_GROUP[ITER4].PRODUCTION	:=	STRING_TO_BOOL(MID(Buff2,FIND(Buff2,'$R')-1,1));
					6:
						TBL_GROUP[ITER4].PROGRAMMATION	:=	STRING_TO_BOOL(MID(Buff2,FIND(Buff2,'$R')-1,1));
					7:
						TBL_GROUP[ITER4].SUPERVISEUR	:=	STRING_TO_BOOL(MID(Buff2,FIND(Buff2,'$R')-1,1));
					8:
						TBL_GROUP[ITER4].CONF_TRF	:=	STRING_TO_BOOL(MID(Buff2,FIND(Buff2,'$R')-1,1));
					9:
						TBL_GROUP[ITER4].MODIF_ENLIGNE	:=	STRING_TO_BOOL(MID(Buff2,FIND(Buff2,'$R')-1,1));
					10:
						TBL_GROUP[ITER4].ARCHIVE_EV	:=	STRING_TO_BOOL(MID(Buff2,FIND(Buff2,'$R')-1,1));
					11:
						TBL_GROUP[ITER4].DECONSIGNATION	:=	STRING_TO_BOOL(MID(Buff2,FIND(Buff2,'$R')-1,1));

				END_CASE
			END_IF
			Step2 := 3;
		ELSE
			IF ITER3 > 5 AND ITER4 <= 30 THEN
				ITER3 := 1;
				ITER4 := ITER4 + 1;
				Step2 := 3;
				TBL_USER[ITER4-NB_GROUP].GROUPE			:=	MID(Buff2,FIND(Buff2,'$R')-1,1);
			ELSE
				IF ITER4 > 30 THEN
					Step2 := 50;
				ELSE
					CASE ITER3 OF
						1:
							TBL_USER[ITER4-NB_GROUP].GROUPE			:=	MID(Buff2,FIND(Buff2,'$R')-1,1);
						2:
							TBL_USER[ITER4-NB_GROUP].LOGIN			:=	MID(Buff2,FIND(Buff2,'$R')-1,1);
						3:
							TBL_USER[ITER4-NB_GROUP].NOM			:=	MID(Buff2,FIND(Buff2,'$R')-1,1);
						4:
							TBL_USER[ITER4-NB_GROUP].PASS			:=	MID(Buff2,FIND(Buff2,'$R')-1,1);
						5:
							TBL_USER[ITER4-NB_GROUP].PRENOM		:=	MID(Buff2,FIND(Buff2,'$R')-1,1);
					END_CASE
					Step2 := 3;
				END_IF
			END_IF
		END_IF
		ITER3 := ITER3 + 1;

	30:
		FCT_Ferm_File( bExecute := FALSE );
		FCT_Ferm_File( 	sNetId:='',
				hFile:=hDestFile,
				bExecute:=TRUE,
				tTimeout:=T#10s  );
		Step2 := Step2 + 1;

	31:
		FCT_Ferm_File( bExecute := FALSE );
		IF ( NOT FCT_Ferm_File.bBusy ) THEN
			IF ( FCT_Ferm_File.bError ) THEN
				ADSLOGSTR( msgCtrlMask := ADSLOG_MSGTYPE_ERROR ,
        				msgFmtStr :=  'Error Code 12', strArg := ''); (* Erreur de fermeture du fichier. *)
			ELSE
				ADSLOGSTR( msgCtrlMask := ADSLOG_MSGTYPE_MSGBOX,
        				msgFmtStr :=  'OK !', strArg := '');
				RQ_SAV_PERSISTENT	:=	TRUE;		(*Ecriture des variables persistante*)
			END_IF
			Step2 := 50;
			hDestFile := 0;
		END_IF

	50:
		IF ( hDestFile <> 0 ) THEN
			Step2 := 30; (* close the destination file*)
		ELSE
			Step2	:=	0;
		END_IF
END_CASE
(*===================================================================================================*)

IF Step > 0 THEN
	SAVE_EC	:=	TRUE;
ELSE
	SAVE_EC	:=	FALSE;
END_IF

IF Step2 > 0 THEN
	LOAD_EC	:=	TRUE;
ELSE
	LOAD_EC	:=	FALSE;
END_IF

IF TBL_GROUP[NB_GROUP].NOM	<>	'' THEN
	STOP_GROUP	:=	TRUE;
ELSE
	STOP_GROUP	:=	FALSE;
END_IF

IF TBL_USER[NB_USER].LOGIN	<>	'' THEN
	STOP_USER	:=	TRUE;
ELSE
	STOP_USER	:=	FALSE;
END_IF

(*********************************************************** Autorisation modification groupe **********************************************************)
IF TBL_GROUP[LIGNE_GROUP].NOM = '' THEN
	AUT_MOD_GRP		:=	FALSE;
ELSE
	AUT_MOD_GRP		:=	TRUE;
END_IF
(*==============================================================================================*)

(*********************************************************** Autorisation modification utilisateur **********************************************************)
IF TBL_USER[LIGNE].LOGIN = '' THEN
	AUT_MOD_USER		:=	FALSE;
ELSE
	AUT_MOD_USER		:=	TRUE;
END_IF
(*==============================================================================================*)


(****************************************************** 	Organisation des groupes après suppression **********************************************)
IF DD_ORG_GRP THEN

